LIN {X 0,Y 421.13,Z 404.126,A -85,B 0,C 180,E1 -10185.61,E2 -10185.61} C_VEL
LIN {X 0,Y 421.83,Z 391.614,A -85,B 0,C 180,E1 -10186.266,E2 -10186.266} C_VEL
LIN {X 0,Y 422.346,Z 378.565,A -85,B 0,C 180,E1 -10186.743,E2 -10186.743} C_VEL
LIN {X 0,Y 422.673,Z 363.001,A -85,B 0,C 180,E1 -10187.072,E2 -10187.072} C_VEL
LIN {X 0,Y 423.413,Z 291.136,A -85,B 0,C 180,E1 -10188.331,E2 -10188.331} C_VEL
LIN {X 0,Y 419.56,Z 265.858,A -85,B 0,C 180,E1 -10188.963,E2 -10188.963} C_VEL
LIN {X 0,Y 420.642,Z 248.412,A -85,B 0,C 180,E1 -10192.339,E2 -10192.339} C_VEL
LIN {X 0,Y 421.257,Z 237.979,A -85,B 0,C 180,E1 -10194.387,E2 -10194.387} C_VEL
LIN {X 0,Y 419.001,Z 226.058,A -85,B 0,C 180,E1 -10196.928,E2 -10196.928} C_VEL
LIN {X 0,Y 418.244,Z 222.39,A -85,B 0,C 180,E1 -10197.752,E2 -10197.752} C_VEL
LIN {X 0,Y 418.218,Z 222.388,A -85,B 0,C 180,E1 -10201.01,E2 -10201.01} C_VEL
LIN {X 0,Y 418.219,Z 222.392,A -85,B 0,C 180,E1 -10203.679,E2 -10203.679} C_VEL
LIN {X 0,Y 418.234,Z 222.385,A -85,B 0,C 180,E1 -10207.224,E2 -10207.224} C_VEL
LIN {X 0,Y 418.214,Z 222.386,A -85,B 0,C 180,E1 -10210.948,E2 -10210.948} C_VEL
LIN {X 0,Y 418.164,Z 222.4,A -85,B 0,C 180,E1 -10213.719,E2 -10213.719} C_VEL
LIN {X 0,Y 418.184,Z 222.391,A -85,B 0,C 180,E1 -10216.441,E2 -10216.441} C_VEL
LIN {X 0,Y 418.213,Z 222.388,A -85,B 0,C 180,E1 -10219.13,E2 -10219.13} C_VEL
LIN {X 0,Y 418.23,Z 222.384,A -85,B 0,C 180,E1 -10222.771,E2 -10222.771} C_VEL
LIN {X 0,Y 418.223,Z 222.386,A -85,B 0,C 180,E1 -10226.316,E2 -10226.316} C_VEL
LIN {X 0,Y 418.237,Z 222.39,A -85,B 0,C 180,E1 -10229.723,E2 -10229.723} C_VEL
LIN {X 0,Y 418.197,Z 222.389,A -85,B 0,C 180,E1 -10233.011,E2 -10233.011} C_VEL
LIN {X 0,Y 418.255,Z 222.382,A -85,B 0,C 180,E1 -10236.212,E2 -10236.212} C_VEL
LIN {X 0,Y 418.237,Z 222.387,A -85,B 0,C 180,E1 -10239.332,E2 -10239.332} C_VEL
LIN {X 0,Y 418.261,Z 222.381,A -85,B 0,C 180,E1 -10242.39,E2 -10242.39} C_VEL
LIN {X 0,Y 418.28,Z 222.383,A -85,B 0,C 180,E1 -10245.397,E2 -10245.397} C_VEL
LIN {X 0,Y 418.291,Z 222.377,A -85,B 0,C 180,E1 -10248.363,E2 -10248.363} C_VEL
LIN {X 0,Y 418.441,Z 222.358,A -85,B 0,C 180,E1 -10252.273,E2 -10252.273} C_VEL
LIN {X 0,Y 418.46,Z 222.356,A -85,B 0,C 180,E1 -10254.211,E2 -10254.211} C_VEL
LIN {X 0,Y 418.518,Z 222.35,A -85,B 0,C 180,E1 -10258.07,E2 -10258.07} C_VEL
LIN {X 0,Y 418.393,Z 222.365,A -85,B 0,C 180,E1 -10260.957,E2 -10260.957} C_VEL
LIN {X 0,Y 418.465,Z 222.356,A -85,B 0,C 180,E1 -10262.882,E2 -10262.882} C_VEL
LIN {X 0,Y 418.418,Z 222.361,A -85,B 0,C 180,E1 -10266.746,E2 -10266.746} C_VEL
LIN {X 0,Y 418.307,Z 222.379,A -85,B 0,C 180,E1 -10269.666,E2 -10269.666} C_VEL
LIN {X 0,Y 418.326,Z 222.375,A -85,B 0,C 180,E1 -10272.994,E2 -10272.994} C_VEL
LIN {X 0,Y 418.288,Z 222.378,A -85,B 0,C 180,E1 -10276.729,E2 -10276.729} C_VEL
LIN {X 0,Y 418.244,Z 222.385,A -85,B 0,C 180,E1 -10279.784,E2 -10279.784} C_VEL
LIN {X 0,Y 418.208,Z 222.388,A -85,B 0,C 180,E1 -10282.731,E2 -10282.731} C_VEL
LIN {X 0,Y 418.208,Z 222.389,A -85,B 0,C 180,E1 -10285.9,E2 -10285.9} C_VEL
LIN {X 0,Y 418.231,Z 222.389,A -85,B 0,C 180,E1 -10289.156,E2 -10289.156} C_VEL
LIN {X 0,Y 418.22,Z 222.387,A -85,B 0,C 180,E1 -10292.838,E2 -10292.838} C_VEL
LIN {X 0,Y 418.204,Z 222.387,A -85,B 0,C 180,E1 -10296.232,E2 -10296.232} C_VEL
LIN {X 0,Y 418.208,Z 222.39,A -85,B 0,C 180,E1 -10299.677,E2 -10299.677} C_VEL
LIN {X 0,Y 418.186,Z 222.39,A -85,B 0,C 180,E1 -10302.316,E2 -10302.316} C_VEL
LIN {X 0,Y 418.191,Z 222.394,A -85,B 0,C 180,E1 -10305.104,E2 -10305.104} C_VEL
LIN {X 0,Y 418.191,Z 222.391,A -85,B 0,C 180,E1 -10307.762,E2 -10307.762} C_VEL
LIN {X 0,Y 418.206,Z 222.391,A -85,B 0,C 180,E1 -10311.554,E2 -10311.554} C_VEL
LIN {X 0,Y 418.207,Z 222.394,A -85,B 0,C 180,E1 -10315.155,E2 -10315.155} C_VEL
LIN {X 0,Y 418.191,Z 222.393,A -85,B 0,C 180,E1 -10317.468,E2 -10317.468} C_VEL
LIN {X 0,Y 418.22,Z 222.389,A -85,B 0,C 180,E1 -10320.89,E2 -10320.89} C_VEL
LIN {X 0,Y 418.216,Z 222.386,A -85,B 0,C 180,E1 -10324.093,E2 -10324.093} C_VEL
LIN {X 0,Y 418.218,Z 222.389,A -85,B 0,C 180,E1 -10327.534,E2 -10327.534} C_VEL
LIN {X 0,Y 418.257,Z 222.381,A -85,B 0,C 180,E1 -10330.363,E2 -10330.363} C_VEL
LIN {X 0,Y 418.265,Z 222.384,A -85,B 0,C 180,E1 -10333.403,E2 -10333.403} C_VEL
LIN {X 0,Y 418.293,Z 222.382,A -85,B 0,C 180,E1 -10336.992,E2 -10336.992} C_VEL
LIN {X 0,Y 418.305,Z 222.375,A -85,B 0,C 180,E1 -10340.328,E2 -10340.328} C_VEL
LIN {X 0,Y 418.453,Z 222.362,A -85,B 0,C 180,E1 -10343.248,E2 -10343.248} C_VEL
LIN {X 0,Y 418.286,Z 222.383,A -85,B 0,C 180,E1 -10345.181,E2 -10345.181} C_VEL
LIN {X 0,Y 418.482,Z 222.353,A -85,B 0,C 180,E1 -10348.075,E2 -10348.075} C_VEL
LIN {X 0,Y 418.61,Z 222.337,A -85,B 0,C 180,E1 -10350,E2 -10350} C_VEL
LIN {X 0,Y 418.456,Z 222.362,A -85,B 0,C 180,E1 -10352.888,E2 -10352.888} C_VEL
LIN {X 0,Y 418.479,Z 222.355,A -85,B 0,C 180,E1 -10355.783,E2 -10355.783} C_VEL
LIN {X 0,Y 418.355,Z 222.375,A -85,B 0,C 180,E1 -10358.696,E2 -10358.696} C_VEL
LIN {X 0,Y 418.317,Z 222.57,A -85,B 0,C 180,E1 -10360.772,E2 -10360.772} C_VEL
LIN {X 0,Y 419.131,Z 226.7,A -85,B 0,C 180,E1 -10361.775,E2 -10361.775} C_VEL
LIN {X 0,Y 418.75,Z 229.04,A -85,B 0,C 180,E1 -10362.288,E2 -10362.288} C_VEL
LIN {X 0,Y 416.077,Z 233.116,A -85,B 0,C 180,E1 -10363.077,E2 -10363.077} C_VEL
LIN {X 0,Y 413.78,Z 237.058,A -85,B 0,C 180,E1 -10363.687,E2 -10363.687} C_VEL
LIN {X 0,Y 413.53,Z 239.678,A -85,B 0,C 180,E1 -10363.885,E2 -10363.885} C_VEL
LIN {X 0,Y 413.619,Z 240.251,A -85,B 0,C 180,E1 -10363.905,E2 -10363.905} C_VEL
LIN {X 0,Y 417.073,Z 257.796,A -85,B 0,C 180,E1 -10364.388,E2 -10364.388} C_VEL
LIN {X 0,Y 415.839,Z 344.239,A -85,B 0,C 180,E1 -10365.94,E2 -10365.94} C_VEL
LIN {X 0,Y 415.403,Z 357.444,A -85,B 0,C 180,E1 -10366.367,E2 -10366.367} C_VEL
LIN {X 0,Y 414.936,Z 370.256,A -85,B 0,C 180,E1 -10366.988,E2 -10366.988} C_VEL
LIN {X 0,Y 414.351,Z 382.19,A -85,B 0,C 180,E1 -10367.776,E2 -10367.776} C_VEL
LIN {X 0,Y 413.625,Z 393.478,A -85,B 0,C 180,E1 -10368.735,E2 -10368.735} C_VEL
LIN {X 0,Y 412.878,Z 404.419,A -85,B 0,C 180,E1 -10369.903,E2 -10369.903} C_VEL
LIN {X 0,Y 412.209,Z 412.623,A -85,B 0,C 180,E1 -10370.979,E2 -10370.979} C_VEL
LIN {X 0,Y 411.605,Z 421.45,A -85,B 0,C 180,E1 -10372.403,E2 -10372.403} C_VEL
LIN {X 0,Y 411.011,Z 429.216,A -85,B 0,C 180,E1 -10373.96,E2 -10373.96} C_VEL
LIN {X 0,Y 410.626,Z 434.689,A -85,B 0,C 180,E1 -10375.333,E2 -10375.333} C_VEL
LIN {X 0,Y 410.322,Z 440.075,A -85,B 0,C 180,E1 -10377.063,E2 -10377.063} C_VEL
LIN {X 0,Y 410.119,Z 443.73,A -85,B 0,C 180,E1 -10378.673,E2 -10378.673} C_VEL
LIN {X 0,Y 409.947,Z 445.615,A -85,B 0,C 180,E1 -10379.812,E2 -10379.812} C_VEL
LIN {X 0,Y 409.835,Z 446.965,A -85,B 0,C 180,E1 -10380.989,E2 -10380.989} C_VEL
LIN {X 0,Y 409.79,Z 447.919,A -85,B 0,C 180,E1 -10382.837,E2 -10382.837} C_VEL
LIN {X 0,Y 409.805,Z 447.533,A -85,B 0,C 180,E1 -10384.61,E2 -10384.61} C_VEL
LIN {X 0,Y 409.934,Z 445.905,A -85,B 0,C 180,E1 -10386.329,E2 -10386.329} C_VEL
LIN {X 0,Y 410.214,Z 442.914,A -85,B 0,C 180,E1 -10388.079,E2 -10388.079} C_VEL
LIN {X 0,Y 410.418,Z 439.178,A -85,B 0,C 180,E1 -10389.607,E2 -10389.607} C_VEL
LIN {X 0,Y 410.771,Z 434.092,A -85,B 0,C 180,E1 -10391.178,E2 -10391.178} C_VEL
LIN {X 0,Y 411.289,Z 427.699,A -85,B 0,C 180,E1 -10392.724,E2 -10392.724} C_VEL
LIN {X 0,Y 411.967,Z 419.754,A -85,B 0,C 180,E1 -10394.245,E2 -10394.245} C_VEL
LIN {X 0,Y 412.732,Z 410.523,A -85,B 0,C 180,E1 -10395.656,E2 -10395.656} C_VEL
LIN {X 0,Y 413.412,Z 401.414,A -85,B 0,C 180,E1 -10396.79,E2 -10396.79} C_VEL
LIN {X 0,Y 414.188,Z 391.232,A -85,B 0,C 180,E1 -10397.822,E2 -10397.822} C_VEL
LIN {X 0,Y 414.926,Z 379.902,A -85,B 0,C 180,E1 -10398.732,E2 -10398.732} C_VEL
LIN {X 0,Y 415.566,Z 367.793,A -85,B 0,C 180,E1 -10399.483,E2 -10399.483} C_VEL
LIN {X 0,Y 416.066,Z 355.316,A -85,B 0,C 180,E1 -10400.051,E2 -10400.051} C_VEL
LIN {X 0,Y 416.391,Z 342.292,A -85,B 0,C 180,E1 -10400.433,E2 -10400.433} C_VEL
LIN {X 0,Y 417.621,Z 257.355,A -85,B 0,C 180,E1 -10401.968,E2 -10401.968} C_VEL
LIN {X 0,Y 413.763,Z 239.192,A -85,B 0,C 180,E1 -10402.513,E2 -10402.513} C_VEL
LIN {X 0,Y 413.33,Z 237.054,A -85,B 0,C 180,E1 -10402.61,E2 -10402.61} C_VEL
LIN {X 0,Y 413.225,Z 233.046,A -85,B 0,C 180,E1 -10403.478,E2 -10403.478} C_VEL
LIN {X 0,Y 411.22,Z 223.265,A -85,B 0,C 180,E1 -10405.751,E2 -10405.751} C_VEL
LIN {X 0,Y 411.162,Z 223.272,A -85,B 0,C 180,E1 -10409.159,E2 -10409.159} C_VEL
LIN {X 0,Y 411.228,Z 223.26,A -85,B 0,C 180,E1 -10412.528,E2 -10412.528} C_VEL
LIN {X 0,Y 411.197,Z 223.263,A -85,B 0,C 180,E1 -10415.79,E2 -10415.79} C_VEL
LIN {X 0,Y 411.169,Z 223.273,A -85,B 0,C 180,E1 -10418.972,E2 -10418.972} C_VEL
LIN {X 0,Y 411.228,Z 223.261,A -85,B 0,C 180,E1 -10422.091,E2 -10422.091} C_VEL
LIN {X 0,Y 411.239,Z 223.259,A -85,B 0,C 180,E1 -10425.153,E2 -10425.153} C_VEL
LIN {X 0,Y 411.28,Z 223.251,A -85,B 0,C 180,E1 -10428.174,E2 -10428.174} C_VEL
LIN {X 0,Y 411.422,Z 223.232,A -85,B 0,C 180,E1 -10432.197,E2 -10432.197} C_VEL
LIN {X 0,Y 411.432,Z 223.233,A -85,B 0,C 180,E1 -10434.123,E2 -10434.123} C_VEL
LIN {X 0,Y 411.498,Z 223.222,A -85,B 0,C 180,E1 -10438.048,E2 -10438.048} C_VEL
LIN {X 0,Y 411.625,Z 223.208,A -85,B 0,C 180,E1 -10440.006,E2 -10440.006} C_VEL
LIN {X 0,Y 411.425,Z 223.235,A -85,B 0,C 180,E1 -10442.943,E2 -10442.943} C_VEL
LIN {X 0,Y 411.424,Z 223.235,A -85,B 0,C 180,E1 -10446.873,E2 -10446.873} C_VEL
LIN {X 0,Y 411.278,Z 223.247,A -85,B 0,C 180,E1 -10449.844,E2 -10449.844} C_VEL
LIN {X 0,Y 411.302,Z 223.247,A -85,B 0,C 180,E1 -10453.109,E2 -10453.109} C_VEL
LIN {X 0,Y 411.257,Z 223.256,A -85,B 0,C 180,E1 -10456.894,E2 -10456.894} C_VEL
LIN {X 0,Y 411.232,Z 223.257,A -85,B 0,C 180,E1 -10459.991,E2 -10459.991} C_VEL
LIN {X 0,Y 411.188,Z 223.262,A -85,B 0,C 180,E1 -10463.153,E2 -10463.153} C_VEL
LIN {X 0,Y 411.167,Z 223.265,A -85,B 0,C 180,E1 -10466.39,E2 -10466.39} C_VEL
LIN {X 0,Y 411.2,Z 223.259,A -85,B 0,C 180,E1 -10469.717,E2 -10469.717} C_VEL
LIN {X 0,Y 411.209,Z 223.257,A -85,B 0,C 180,E1 -10473.16,E2 -10473.16} C_VEL
LIN {X 0,Y 411.194,Z 223.264,A -85,B 0,C 180,E1 -10476.555,E2 -10476.555} C_VEL
LIN {X 0,Y 411.169,Z 223.265,A -85,B 0,C 180,E1 -10479.722,E2 -10479.722} C_VEL
LIN {X 0,Y 411.131,Z 223.273,A -85,B 0,C 180,E1 -10483.144,E2 -10483.144} C_VEL
LIN {X 0,Y 411.156,Z 223.272,A -85,B 0,C 180,E1 -10485.887,E2 -10485.887} C_VEL
LIN {X 0,Y 411.164,Z 223.267,A -85,B 0,C 180,E1 -10489.495,E2 -10489.495} C_VEL
LIN {X 0,Y 411.185,Z 223.269,A -85,B 0,C 180,E1 -10492.027,E2 -10492.027} C_VEL
LIN {X 0,Y 411.208,Z 223.262,A -85,B 0,C 180,E1 -10495.127,E2 -10495.127} C_VEL
LIN {X 0,Y 411.163,Z 223.276,A -85,B 0,C 180,E1 -10498.004,E2 -10498.004} C_VEL
LIN {X 0,Y 411.183,Z 223.271,A -85,B 0,C 180,E1 -10501.408,E2 -10501.408} C_VEL
LIN {X 0,Y 411.184,Z 223.35,A -85,B 0,C 180,E1 -10502.034,E2 -10502.034} C_VEL
LIN {X 0,Y 413.567,Z 234.523,A -85,B 0,C 180,E1 -10504.482,E2 -10504.482} C_VEL
LIN {X 0,Y 414.356,Z 240.401,A -85,B 0,C 180,E1 -10505.714,E2 -10505.714} C_VEL
LIN {X 0,Y 413.278,Z 256.322,A -85,B 0,C 180,E1 -10508.816,E2 -10508.816} C_VEL
LIN {X 0,Y 412.823,Z 264.691,A -85,B 0,C 180,E1 -10510.435,E2 -10510.435} C_VEL
LIN {X 0,Y 416.982,Z 290.686,A -85,B 0,C 180,E1 -10511.14,E2 -10511.14} C_VEL
LIN {X 0,Y 417.212,Z 298.733,A -85,B 0,C 180,E1 -10511.302,E2 -10511.302} C_VEL
LIN {X 0,Y 416.178,Z 374.289,A -85,B 0,C 180,E1 -10512.685,E2 -10512.685} C_VEL
LIN {X 0,Y 415.578,Z 387.154,A -85,B 0,C 180,E1 -10513.103,E2 -10513.103} C_VEL
LIN {X 0,Y 414.874,Z 399.702,A -85,B 0,C 180,E1 -10513.706,E2 -10513.706} C_VEL
LIN {X 0,Y 414.051,Z 411.72,A -85,B 0,C 180,E1 -10514.495,E2 -10514.495} C_VEL
LIN {X 0,Y 413.284,Z 423.495,A -85,B 0,C 180,E1 -10515.499,E2 -10515.499} C_VEL
LIN {X 0,Y 412.488,Z 433.635,A -85,B 0,C 180,E1 -10516.577,E2 -10516.577} C_VEL
LIN {X 0,Y 411.885,Z 442.149,A -85,B 0,C 180,E1 -10517.685,E2 -10517.685} C_VEL
LIN {X 0,Y 411.061,Z 451.381,A -85,B 0,C 180,E1 -10519.16,E2 -10519.16} C_VEL
LIN {X 0,Y 410.606,Z 458.83,A -85,B 0,C 180,E1 -10520.642,E2 -10520.642} C_VEL
LIN {X 0,Y 410.279,Z 464.815,A -85,B 0,C 180,E1 -10522.124,E2 -10522.124} C_VEL
LIN {X 0,Y 410.036,Z 470.092,A -85,B 0,C 180,E1 -10523.803,E2 -10523.803} C_VEL
LIN {X 0,Y 410.016,Z 473.156,A -85,B 0,C 180,E1 -10525.084,E2 -10525.084} C_VEL
LIN {X 0,Y 409.938,Z 475.002,A -85,B 0,C 180,E1 -10526.068,E2 -10526.068} C_VEL
LIN {X 0,Y 410.003,Z 477.393,A -85,B 0,C 180,E1 -10528.035,E2 -10528.035} C_VEL
LIN {X 0,Y 409.945,Z 477.993,A -85,B 0,C 180,E1 -10529.018,E2 -10529.018} C_VEL
LIN {X 0,Y 409.935,Z 478.174,A -85,B 0,C 180,E1 -10530,E2 -10530} C_VEL
LIN {X 0,Y 410.003,Z 477.303,A -85,B 0,C 180,E1 -10531.965,E2 -10531.965} C_VEL
LIN {X 0,Y 409.937,Z 476.274,A -85,B 0,C 180,E1 -10532.948,E2 -10532.948} C_VEL
LIN {X 0,Y 409.938,Z 474.809,A -85,B 0,C 180,E1 -10533.932,E2 -10533.932} C_VEL
LIN {X 0,Y 409.996,Z 471.793,A -85,B 0,C 180,E1 -10535.41,E2 -10535.41} C_VEL
LIN {X 0,Y 410.175,Z 467.711,A -85,B 0,C 180,E1 -10536.888,E2 -10536.888} C_VEL
LIN {X 0,Y 410.432,Z 461.424,A -85,B 0,C 180,E1 -10538.617,E2 -10538.617} C_VEL
LIN {X 0,Y 410.839,Z 454.576,A -85,B 0,C 180,E1 -10540.098,E2 -10540.098} C_VEL
LIN {X 0,Y 411.291,Z 447.586,A -85,B 0,C 180,E1 -10541.333,E2 -10541.333} C_VEL
LIN {X 0,Y 411.942,Z 439.171,A -85,B 0,C 180,E1 -10542.563,E2 -10542.563} C_VEL
LIN {X 0,Y 412.67,Z 428.8,A -85,B 0,C 180,E1 -10543.793,E2 -10543.793} C_VEL
LIN {X 0,Y 413.416,Z 417.096,A -85,B 0,C 180,E1 -10544.899,E2 -10544.899} C_VEL
LIN {X 0,Y 414.136,Z 405.504,A -85,B 0,C 180,E1 -10545.755,E2 -10545.755} C_VEL
LIN {X 0,Y 414.84,Z 393.49,A -85,B 0,C 180,E1 -10546.422,E2 -10546.422} C_VEL
LIN {X 0,Y 415.45,Z 380.532,A -85,B 0,C 180,E1 -10546.934,E2 -10546.934} C_VEL
LIN {X 0,Y 415.772,Z 368.445,A -85,B 0,C 180,E1 -10547.237,E2 -10547.237} C_VEL
LIN {X 0,Y 416.664,Z 292.238,A -85,B 0,C 180,E1 -10548.594,E2 -10548.594} C_VEL
LIN {X 0,Y 412.611,Z 265.599,A -85,B 0,C 180,E1 -10549.276,E2 -10549.276} C_VEL
LIN {X 0,Y 413.796,Z 248.074,A -85,B 0,C 180,E1 -10552.73,E2 -10552.73} C_VEL
LIN {X 0,Y 414.263,Z 238.927,A -85,B 0,C 180,E1 -10554.559,E2 -10554.559} C_VEL
LIN {X 0,Y 411.887,Z 226.556,A -85,B 0,C 180,E1 -10557.25,E2 -10557.25} C_VEL
LIN {X 0,Y 411.196,Z 223.266,A -85,B 0,C 180,E1 -10558.035,E2 -10558.035} C_VEL
LIN {X 0,Y 411.164,Z 223.268,A -85,B 0,C 180,E1 -10561.274,E2 -10561.274} C_VEL
LIN {X 0,Y 411.169,Z 223.265,A -85,B 0,C 180,E1 -10564.336,E2 -10564.336} C_VEL
LIN {X 0,Y 411.187,Z 223.262,A -85,B 0,C 180,E1 -10566.741,E2 -10566.741} C_VEL
LIN {X 0,Y 411.171,Z 223.27,A -85,B 0,C 180,E1 -10569.716,E2 -10569.716} C_VEL
LIN {X 0,Y 411.113,Z 223.272,A -85,B 0,C 180,E1 -10573.14,E2 -10573.14} C_VEL
LIN {X 0,Y 411.151,Z 223.272,A -85,B 0,C 180,E1 -10575.882,E2 -10575.882} C_VEL
LIN {X 0,Y 411.163,Z 223.269,A -85,B 0,C 180,E1 -10579.489,E2 -10579.489} C_VEL
LIN {X 0,Y 411.18,Z 223.266,A -85,B 0,C 180,E1 -10582.02,E2 -10582.02} C_VEL
LIN {X 0,Y 411.191,Z 223.262,A -85,B 0,C 180,E1 -10585.123,E2 -10585.123} C_VEL
LIN {X 0,Y 411.157,Z 223.269,A -85,B 0,C 180,E1 -10587.998,E2 -10587.998} C_VEL
LIN {X 0,Y 411.17,Z 223.268,A -85,B 0,C 180,E1 -10591.402,E2 -10591.402} C_VEL
LIN {X 0,Y 411.19,Z 223.262,A -85,B 0,C 180,E1 -10594.937,E2 -10594.937} C_VEL
LIN {X 0,Y 411.201,Z 223.264,A -85,B 0,C 180,E1 -10597.909,E2 -10597.909} C_VEL
LIN {X 0,Y 411.187,Z 223.263,A -85,B 0,C 180,E1 -10601.045,E2 -10601.045} C_VEL
LIN {X 0,Y 411.238,Z 223.257,A -85,B 0,C 180,E1 -10604.126,E2 -10604.126} C_VEL
LIN {X 0,Y 411.298,Z 223.25,A -85,B 0,C 180,E1 -10607.161,E2 -10607.161} C_VEL
LIN {X 0,Y 411.265,Z 223.253,A -85,B 0,C 180,E1 -10610.156,E2 -10610.156} C_VEL
LIN {X 0,Y 411.383,Z 223.24,A -85,B 0,C 180,E1 -10613.127,E2 -10613.127} C_VEL
LIN {X 0,Y 411.272,Z 223.253,A -85,B 0,C 180,E1 -10615.093,E2 -10615.093} C_VEL
LIN {X 0,Y 411.487,Z 223.226,A -85,B 0,C 180,E1 -10618.037,E2 -10618.037} C_VEL
LIN {X 0,Y 411.492,Z 223.226,A -85,B 0,C 180,E1 -10621.952,E2 -10621.952} C_VEL
LIN {X 0,Y 411.364,Z 223.239,A -85,B 0,C 180,E1 -10626.5,E2 -10626.5} C_VEL
LIN {X 0,Y 411.291,Z 223.25,A -85,B 0,C 180,E1 -10628.84,E2 -10628.84} C_VEL
LIN {X 0,Y 411.26,Z 223.255,A -85,B 0,C 180,E1 -10631.827,E2 -10631.827} C_VEL
LIN {X 0,Y 411.234,Z 223.257,A -85,B 0,C 180,E1 -10634.847,E2 -10634.847} C_VEL
LIN {X 0,Y 411.22,Z 223.259,A -85,B 0,C 180,E1 -10637.91,E2 -10637.91} C_VEL
LIN {X 0,Y 411.169,Z 223.267,A -85,B 0,C 180,E1 -10641.028,E2 -10641.028} C_VEL
LIN {X 0,Y 411.179,Z 223.263,A -85,B 0,C 180,E1 -10644.211,E2 -10644.211} C_VEL
LIN {X 0,Y 411.21,Z 223.265,A -85,B 0,C 180,E1 -10647.473,E2 -10647.473} C_VEL
LIN {X 0,Y 411.154,Z 223.267,A -85,B 0,C 180,E1 -10650.842,E2 -10650.842} C_VEL
LIN {X 0,Y 411.167,Z 223.264,A -85,B 0,C 180,E1 -10654.328,E2 -10654.328} C_VEL
LIN {X 0,Y 411.154,Z 223.267,A -85,B 0,C 180,E1 -10657.968,E2 -10657.968} C_VEL
LIN {X 0,Y 411.139,Z 223.268,A -85,B 0,C 180,E1 -10660.499,E2 -10660.499} C_VEL
LIN {X 0,Y 411.132,Z 223.274,A -85,B 0,C 180,E1 -10663.128,E2 -10663.128} C_VEL
LIN {X 0,Y 411.121,Z 223.271,A -85,B 0,C 180,E1 -10665.876,E2 -10665.876} C_VEL
LIN {X 0,Y 411.114,Z 223.273,A -85,B 0,C 180,E1 -10668.767,E2 -10668.767} C_VEL
LIN {X 0,Y 411.148,Z 223.267,A -85,B 0,C 180,E1 -10672.022,E2 -10672.022} C_VEL
LIN {X 0,Y 411.152,Z 223.268,A -85,B 0,C 180,E1 -10675.662,E2 -10675.662} C_VEL
LIN {X 0,Y 411.142,Z 223.274,A -85,B 0,C 180,E1 -10679.149,E2 -10679.149} C_VEL
LIN {X 0,Y 411.203,Z 223.26,A -85,B 0,C 180,E1 -10682.519,E2 -10682.519} C_VEL
LIN {X 0,Y 411.173,Z 223.264,A -85,B 0,C 180,E1 -10685.782,E2 -10685.782} C_VEL
LIN {X 0,Y 411.179,Z 223.268,A -85,B 0,C 180,E1 -10688.965,E2 -10688.965} C_VEL
LIN {X 0,Y 411.195,Z 223.261,A -85,B 0,C 180,E1 -10692.083,E2 -10692.083} C_VEL
LIN {X 0,Y 411.205,Z 223.267,A -85,B 0,C 180,E1 -10695.146,E2 -10695.146} C_VEL
LIN {X 0,Y 411.24,Z 223.255,A -85,B 0,C 180,E1 -10698.166,E2 -10698.166} C_VEL
LIN {X 0,Y 411.419,Z 223.233,A -85,B 0,C 180,E1 -10702.146,E2 -10702.146} C_VEL
LIN {X 0,Y 411.438,Z 223.23,A -85,B 0,C 180,E1 -10704.118,E2 -10704.118} C_VEL
LIN {X 0,Y 411.451,Z 223.229,A -85,B 0,C 180,E1 -10708.042,E2 -10708.042} C_VEL
LIN {X 0,Y 411.58,Z 223.213,A -85,B 0,C 180,E1 -10710,E2 -10710} C_VEL
LIN {X 0,Y 411.411,Z 223.24,A -85,B 0,C 180,E1 -10712.937,E2 -10712.937} C_VEL
LIN {X 0,Y 411.438,Z 223.232,A -85,B 0,C 180,E1 -10715.882,E2 -10715.882} C_VEL
LIN {X 0,Y 411.307,Z 223.254,A -85,B 0,C 180,E1 -10718.846,E2 -10718.846} C_VEL
LIN {X 0,Y 411.287,Z 223.317,A -85,B 0,C 180,E1 -10720.522,E2 -10720.522} C_VEL
LIN {X 0,Y 412.947,Z 232.58,A -85,B 0,C 180,E1 -10722.782,E2 -10722.782} C_VEL
LIN {X 0,Y 412.986,Z 237.016,A -85,B 0,C 180,E1 -10723.807,E2 -10723.807} C_VEL
LIN {X 0,Y 413.619,Z 240.251,A -85,B 0,C 180,E1 -10723.905,E2 -10723.905} C_VEL
LIN {X 0,Y 414.059,Z 246.078,A -85,B 0,C 180,E1 -10724.034,E2 -10724.034} C_VEL
LIN {X 0,Y 413.405,Z 251.982,A -85,B 0,C 180,E1 -10724.115,E2 -10724.115} C_VEL
LIN {X 0,Y 410.319,Z 267.779,A -85,B 0,C 180,E1 -10724.271,E2 -10724.271} C_VEL
LIN {X 0,Y 410.095,Z 271.776,A -85,B 0,C 180,E1 -10724.336,E2 -10724.336} C_VEL
LIN {X 0,Y 409.001,Z 345.346,A -85,B 0,C 180,E1 -10725.692,E2 -10725.692} C_VEL
LIN {X 0,Y 408.574,Z 358.46,A -85,B 0,C 180,E1 -10726.135,E2 -10726.135} C_VEL
LIN {X 0,Y 408.079,Z 371.07,A -85,B 0,C 180,E1 -10726.766,E2 -10726.766} C_VEL
LIN {X 0,Y 407.443,Z 382.88,A -85,B 0,C 180,E1 -10727.569,E2 -10727.569} C_VEL
LIN {X 0,Y 406.719,Z 393.807,A -85,B 0,C 180,E1 -10728.516,E2 -10728.516} C_VEL
LIN {X 0,Y 405.976,Z 403.835,A -85,B 0,C 180,E1 -10729.597,E2 -10729.597} C_VEL
LIN {X 0,Y 405.288,Z 412.117,A -85,B 0,C 180,E1 -10730.682,E2 -10730.682} C_VEL
LIN {X 0,Y 404.704,Z 419.962,A -85,B 0,C 180,E1 -10731.923,E2 -10731.923} C_VEL
LIN {X 0,Y 404.18,Z 426.642,A -85,B 0,C 180,E1 -10733.198,E2 -10733.198} C_VEL
LIN {X 0,Y 403.77,Z 433.031,A -85,B 0,C 180,E1 -10734.691,E2 -10734.691} C_VEL
LIN {X 0,Y 403.336,Z 438.668,A -85,B 0,C 180,E1 -10736.38,E2 -10736.38} C_VEL
LIN {X 0,Y 403.146,Z 442.914,A -85,B 0,C 180,E1 -10738.078,E2 -10738.078} C_VEL
LIN {X 0,Y 402.931,Z 445.199,A -85,B 0,C 180,E1 -10739.313,E2 -10739.313} C_VEL
LIN {X 0,Y 402.729,Z 447.451,A -85,B 0,C 180,E1 -10741.246,E2 -10741.246} C_VEL
LIN {X 0,Y 402.705,Z 448.227,A -85,B 0,C 180,E1 -10743.118,E2 -10743.118} C_VEL
LIN {X 0,Y 402.716,Z 447.632,A -85,B 0,C 180,E1 -10744.908,E2 -10744.908} C_VEL
LIN {X 0,Y 402.883,Z 445.816,A -85,B 0,C 180,E1 -10746.651,E2 -10746.651} C_VEL
LIN {X 0,Y 403.152,Z 442.849,A -85,B 0,C 180,E1 -10748.342,E2 -10748.342} C_VEL
LIN {X 0,Y 403.483,Z 438.351,A -85,B 0,C 180,E1 -10750.125,E2 -10750.125} C_VEL
LIN {X 0,Y 403.908,Z 432.676,A -85,B 0,C 180,E1 -10751.789,E2 -10751.789} C_VEL
LIN {X 0,Y 404.565,Z 425.055,A -85,B 0,C 180,E1 -10753.517,E2 -10753.517} C_VEL
LIN {X 0,Y 405.247,Z 417.384,A -85,B 0,C 180,E1 -10754.904,E2 -10754.904} C_VEL
LIN {X 0,Y 405.964,Z 408.684,A -85,B 0,C 180,E1 -10756.185,E2 -10756.185} C_VEL
LIN {X 0,Y 406.884,Z 397.812,A -85,B 0,C 180,E1 -10757.469,E2 -10757.469} C_VEL
LIN {X 0,Y 407.612,Z 387.993,A -85,B 0,C 180,E1 -10758.404,E2 -10758.404} C_VEL
LIN {X 0,Y 408.343,Z 377.279,A -85,B 0,C 180,E1 -10759.223,E2 -10759.223} C_VEL
LIN {X 0,Y 408.928,Z 366.141,A -85,B 0,C 180,E1 -10759.887,E2 -10759.887} C_VEL
LIN {X 0,Y 409.414,Z 353.346,A -85,B 0,C 180,E1 -10760.437,E2 -10760.437} C_VEL
LIN {X 0,Y 409.725,Z 340.434,A -85,B 0,C 180,E1 -10760.792,E2 -10760.792} C_VEL
LIN {X 0,Y 410.991,Z 258.784,A -85,B 0,C 180,E1 -10762.285,E2 -10762.285} C_VEL
LIN {X 0,Y 407.347,Z 241.288,A -85,B 0,C 180,E1 -10762.824,E2 -10762.824} C_VEL
LIN {X 0,Y 406.479,Z 237.409,A -85,B 0,C 180,E1 -10762.964,E2 -10762.964} C_VEL
LIN {X 0,Y 406.045,Z 233.008,A -85,B 0,C 180,E1 -10763.96,E2 -10763.96} C_VEL
LIN {X 0,Y 404.156,Z 224.144,A -85,B 0,C 180,E1 -10766.085,E2 -10766.085} C_VEL
LIN {X 0,Y 404.119,Z 224.148,A -85,B 0,C 180,E1 -10769.721,E2 -10769.721} C_VEL
LIN {X 0,Y 404.164,Z 224.143,A -85,B 0,C 180,E1 -10773.129,E2 -10773.129} C_VEL
LIN {X 0,Y 404.147,Z 224.143,A -85,B 0,C 180,E1 -10775.34,E2 -10775.34} C_VEL
LIN {X 0,Y 404.111,Z 224.147,A -85,B 0,C 180,E1 -10778.586,E2 -10778.586} C_VEL
LIN {X 0,Y 404.185,Z 224.138,A -85,B 0,C 180,E1 -10781.768,E2 -10781.768} C_VEL
LIN {X 0,Y 404.185,Z 224.139,A -85,B 0,C 180,E1 -10784.888,E2 -10784.888} C_VEL
LIN {X 0,Y 404.251,Z 224.126,A -85,B 0,C 180,E1 -10787.965,E2 -10787.965} C_VEL
LIN {X 0,Y 404.25,Z 224.128,A -85,B 0,C 180,E1 -10791.004,E2 -10791.004} C_VEL
LIN {X 0,Y 404.382,Z 224.111,A -85,B 0,C 180,E1 -10794.02,E2 -10794.02} C_VEL
LIN {X 0,Y 404.467,Z 224.098,A -85,B 0,C 180,E1 -10798.014,E2 -10798.014} C_VEL
LIN {X 0,Y 404.594,Z 224.084,A -85,B 0,C 180,E1 -10800.006,E2 -10800.006} C_VEL
LIN {X 0,Y 404.385,Z 224.113,A -85,B 0,C 180,E1 -10802.994,E2 -10802.994} C_VEL
LIN {X 0,Y 404.375,Z 224.114,A -85,B 0,C 180,E1 -10806.993,E2 -10806.993} C_VEL
LIN {X 0,Y 404.242,Z 224.131,A -85,B 0,C 180,E1 -10811.03,E2 -10811.03} C_VEL
LIN {X 0,Y 404.207,Z 224.131,A -85,B 0,C 180,E1 -10814.093,E2 -10814.093} C_VEL
LIN {X 0,Y 404.202,Z 224.132,A -85,B 0,C 180,E1 -10817.197,E2 -10817.197} C_VEL
LIN {X 0,Y 404.165,Z 224.14,A -85,B 0,C 180,E1 -10820.356,E2 -10820.356} C_VEL
LIN {X 0,Y 404.149,Z 224.137,A -85,B 0,C 180,E1 -10823.58,E2 -10823.58} C_VEL
LIN {X 0,Y 404.101,Z 224.146,A -85,B 0,C 180,E1 -10826.888,E2 -10826.888} C_VEL
LIN {X 0,Y 404.147,Z 224.139,A -85,B 0,C 180,E1 -10830.29,E2 -10830.29} C_VEL
LIN {X 0,Y 404.143,Z 224.137,A -85,B 0,C 180,E1 -10833.817,E2 -10833.817} C_VEL
LIN {X 0,Y 404.136,Z 224.142,A -85,B 0,C 180,E1 -10836.877,E2 -10836.877} C_VEL
LIN {X 0,Y 404.125,Z 224.144,A -85,B 0,C 180,E1 -10840.078,E2 -10840.078} C_VEL
LIN {X 0,Y 404.088,Z 224.151,A -85,B 0,C 180,E1 -10843.076,E2 -10843.076} C_VEL
LIN {X 0,Y 404.114,Z 224.15,A -85,B 0,C 180,E1 -10845.923,E2 -10845.923} C_VEL
LIN {X 0,Y 404.106,Z 224.15,A -85,B 0,C 180,E1 -10848.635,E2 -10848.635} C_VEL
LIN {X 0,Y 404.142,Z 224.142,A -85,B 0,C 180,E1 -10851.499,E2 -10851.499} C_VEL
LIN {X 0,Y 404.179,Z 224.139,A -85,B 0,C 180,E1 -10854.985,E2 -10854.985} C_VEL
LIN {X 0,Y 404.141,Z 224.149,A -85,B 0,C 180,E1 -10858.447,E2 -10858.447} C_VEL
LIN {X 0,Y 404.165,Z 224.218,A -85,B 0,C 180,E1 -10861.717,E2 -10861.717} C_VEL
LIN {X 0,Y 406.692,Z 236.252,A -85,B 0,C 180,E1 -10864.405,E2 -10864.405} C_VEL
LIN {X 0,Y 407.447,Z 241.593,A -85,B 0,C 180,E1 -10865.546,E2 -10865.546} C_VEL
LIN {X 0,Y 406.417,Z 256.178,A -85,B 0,C 180,E1 -10868.441,E2 -10868.441} C_VEL
LIN {X 0,Y 405.946,Z 264.397,A -85,B 0,C 180,E1 -10870.06,E2 -10870.06} C_VEL
LIN {X 0,Y 410.164,Z 290.345,A -85,B 0,C 180,E1 -10870.789,E2 -10870.789} C_VEL
LIN {X 0,Y 410.55,Z 295.777,A -85,B 0,C 180,E1 -10870.913,E2 -10870.913} C_VEL
LIN {X 0,Y 409.461,Z 373.623,A -85,B 0,C 180,E1 -10872.36,E2 -10872.36} C_VEL
LIN {X 0,Y 408.849,Z 386.608,A -85,B 0,C 180,E1 -10872.784,E2 -10872.784} C_VEL
LIN {X 0,Y 408.076,Z 399.775,A -85,B 0,C 180,E1 -10873.427,E2 -10873.427} C_VEL
LIN {X 0,Y 407.206,Z 411.685,A -85,B 0,C 180,E1 -10874.227,E2 -10874.227} C_VEL
LIN {X 0,Y 406.397,Z 423.402,A -85,B 0,C 180,E1 -10875.248,E2 -10875.248} C_VEL
LIN {X 0,Y 405.577,Z 433.536,A -85,B 0,C 180,E1 -10876.348,E2 -10876.348} C_VEL
LIN {X 0,Y 404.78,Z 443.633,A -85,B 0,C 180,E1 -10877.72,E2 -10877.72} C_VEL
LIN {X 0,Y 403.951,Z 452.56,A -85,B 0,C 180,E1 -10879.221,E2 -10879.221} C_VEL
LIN {X 0,Y 403.493,Z 459.734,A -85,B 0,C 180,E1 -10880.729,E2 -10880.729} C_VEL
LIN {X 0,Y 403.14,Z 466.288,A -85,B 0,C 180,E1 -10882.487,E2 -10882.487} C_VEL
LIN {X 0,Y 402.913,Z 470.62,A -85,B 0,C 180,E1 -10883.993,E2 -10883.993} C_VEL
LIN {X 0,Y 402.925,Z 472.924,A -85,B 0,C 180,E1 -10884.997,E2 -10884.997} C_VEL
LIN {X 0,Y 402.858,Z 474.761,A -85,B 0,C 180,E1 -10885.999,E2 -10885.999} C_VEL
LIN {X 0,Y 402.914,Z 477.143,A -85,B 0,C 180,E1 -10888.001,E2 -10888.001} C_VEL
LIN {X 0,Y 402.873,Z 477.739,A -85,B 0,C 180,E1 -10889.001,E2 -10889.001} C_VEL
LIN {X 0,Y 402.86,Z 477.909,A -85,B 0,C 180,E1 -10890,E2 -10890} C_VEL
LIN {X 0,Y 402.873,Z 477.663,A -85,B 0,C 180,E1 -10891,E2 -10891} C_VEL
LIN {X 0,Y 402.914,Z 477.027,A -85,B 0,C 180,E1 -10891.999,E2 -10891.999} C_VEL
LIN {X 0,Y 402.837,Z 475.991,A -85,B 0,C 180,E1 -10893,E2 -10893} C_VEL
LIN {X 0,Y 402.858,Z 474.514,A -85,B 0,C 180,E1 -10894.001,E2 -10894.001} C_VEL
LIN {X 0,Y 402.896,Z 471.482,A -85,B 0,C 180,E1 -10895.505,E2 -10895.505} C_VEL
LIN {X 0,Y 403.087,Z 467.384,A -85,B 0,C 180,E1 -10897.01,E2 -10897.01} C_VEL
LIN {X 0,Y 403.384,Z 461.08,A -85,B 0,C 180,E1 -10898.769,E2 -10898.769} C_VEL
LIN {X 0,Y 403.784,Z 454.209,A -85,B 0,C 180,E1 -10900.277,E2 -10900.277} C_VEL
LIN {X 0,Y 404.312,Z 447.199,A -85,B 0,C 180,E1 -10901.531,E2 -10901.531} C_VEL
LIN {X 0,Y 404.953,Z 438.754,A -85,B 0,C 180,E1 -10902.784,E2 -10902.784} C_VEL
LIN {X 0,Y 405.696,Z 428.33,A -85,B 0,C 180,E1 -10904.035,E2 -10904.035} C_VEL
LIN {X 0,Y 406.544,Z 416.585,A -85,B 0,C 180,E1 -10905.157,E2 -10905.157} C_VEL
LIN {X 0,Y 407.284,Z 404.895,A -85,B 0,C 180,E1 -10906.027,E2 -10906.027} C_VEL
LIN {X 0,Y 408.019,Z 392.774,A -85,B 0,C 180,E1 -10906.704,E2 -10906.704} C_VEL
LIN {X 0,Y 408.617,Z 379.633,A -85,B 0,C 180,E1 -10907.226,E2 -10907.226} C_VEL
LIN {X 0,Y 408.953,Z 367.023,A -85,B 0,C 180,E1 -10907.534,E2 -10907.534} C_VEL
LIN {X 0,Y 409.823,Z 292.532,A -85,B 0,C 180,E1 -10908.885,E2 -10908.885} C_VEL
LIN {X 0,Y 405.707,Z 265.348,A -85,B 0,C 180,E1 -10909.597,E2 -10909.597} C_VEL
LIN {X 0,Y 406.921,Z 247.707,A -85,B 0,C 180,E1 -10913.136,E2 -10913.136} C_VEL
LIN {X 0,Y 407.385,Z 241.186,A -85,B 0,C 180,E1 -10914.458,E2 -10914.458} C_VEL
LIN {X 0,Y 405.976,Z 232.952,A -85,B 0,C 180,E1 -10916.258,E2 -10916.258} C_VEL
LIN {X 0,Y 404.141,Z 224.145,A -85,B 0,C 180,E1 -10918.285,E2 -10918.285} C_VEL
LIN {X 0,Y 404.125,Z 224.146,A -85,B 0,C 180,E1 -10921.549,E2 -10921.549} C_VEL
LIN {X 0,Y 404.133,Z 224.141,A -85,B 0,C 180,E1 -10925.02,E2 -10925.02} C_VEL
LIN {X 0,Y 404.137,Z 224.14,A -85,B 0,C 180,E1 -10928.5,E2 -10928.5} C_VEL
LIN {X 0,Y 404.093,Z 224.15,A -85,B 0,C 180,E1 -10931.59,E2 -10931.59} C_VEL
LIN {X 0,Y 404.131,Z 224.145,A -85,B 0,C 180,E1 -10935.479,E2 -10935.479} C_VEL
LIN {X 0,Y 404.105,Z 224.144,A -85,B 0,C 180,E1 -10938.629,E2 -10938.629} C_VEL
LIN {X 0,Y 404.138,Z 224.144,A -85,B 0,C 180,E1 -10941.493,E2 -10941.493} C_VEL
LIN {X 0,Y 404.162,Z 224.137,A -85,B 0,C 180,E1 -10944.977,E2 -10944.977} C_VEL
LIN {X 0,Y 404.139,Z 224.143,A -85,B 0,C 180,E1 -10947.374,E2 -10947.374} C_VEL
LIN {X 0,Y 404.15,Z 224.138,A -85,B 0,C 180,E1 -10950.858,E2 -10950.858} C_VEL
LIN {X 0,Y 404.153,Z 224.138,A -85,B 0,C 180,E1 -10954.719,E2 -10954.719} C_VEL
LIN {X 0,Y 404.167,Z 224.142,A -85,B 0,C 180,E1 -10957.503,E2 -10957.503} C_VEL
LIN {X 0,Y 404.137,Z 224.14,A -85,B 0,C 180,E1 -10960.701,E2 -10960.701} C_VEL
LIN {X 0,Y 404.21,Z 224.135,A -85,B 0,C 180,E1 -10963.843,E2 -10963.843} C_VEL
LIN {X 0,Y 404.281,Z 224.123,A -85,B 0,C 180,E1 -10966.934,E2 -10966.934} C_VEL
LIN {X 0,Y 404.233,Z 224.13,A -85,B 0,C 180,E1 -10969.983,E2 -10969.983} C_VEL
LIN {X 0,Y 404.333,Z 224.117,A -85,B 0,C 180,E1 -10973.006,E2 -10973.006} C_VEL
LIN {X 0,Y 404.244,Z 224.128,A -85,B 0,C 180,E1 -10975.008,E2 -10975.008} C_VEL
LIN {X 0,Y 404.456,Z 224.102,A -85,B 0,C 180,E1 -10978.003,E2 -10978.003} C_VEL
LIN {X 0,Y 404.461,Z 224.101,A -85,B 0,C 180,E1 -10981.986,E2 -10981.986} C_VEL
LIN {X 0,Y 404.317,Z 224.117,A -85,B 0,C 180,E1 -10986.497,E2 -10986.497} C_VEL
LIN {X 0,Y 404.24,Z 224.129,A -85,B 0,C 180,E1 -10988.996,E2 -10988.996} C_VEL
LIN {X 0,Y 404.234,Z 224.129,A -85,B 0,C 180,E1 -10992.036,E2 -10992.036} C_VEL
LIN {X 0,Y 404.18,Z 224.138,A -85,B 0,C 180,E1 -10995.112,E2 -10995.112} C_VEL
LIN {X 0,Y 404.179,Z 224.135,A -85,B 0,C 180,E1 -10998.232,E2 -10998.232} C_VEL
LIN {X 0,Y 404.132,Z 224.148,A -85,B 0,C 180,E1 -11001.412,E2 -11001.412} C_VEL
LIN {X 0,Y 404.133,Z 224.141,A -85,B 0,C 180,E1 -11004.661,E2 -11004.661} C_VEL
LIN {X 0,Y 404.155,Z 224.139,A -85,B 0,C 180,E1 -11007.994,E2 -11007.994} C_VEL
LIN {X 0,Y 404.104,Z 224.149,A -85,B 0,C 180,E1 -11011.552,E2 -11011.552} C_VEL
LIN {X 0,Y 404.146,Z 224.142,A -85,B 0,C 180,E1 -11015.011,E2 -11015.011} C_VEL
LIN {X 0,Y 404.114,Z 224.144,A -85,B 0,C 180,E1 -11018.752,E2 -11018.752} C_VEL
LIN {X 0,Y 404.08,Z 224.151,A -85,B 0,C 180,E1 -11021.594,E2 -11021.594} C_VEL
LIN {X 0,Y 404.102,Z 224.145,A -85,B 0,C 180,E1 -11024.517,E2 -11024.517} C_VEL
LIN {X 0,Y 404.088,Z 224.153,A -85,B 0,C 180,E1 -11027.291,E2 -11027.291} C_VEL
LIN {X 0,Y 404.12,Z 224.142,A -85,B 0,C 180,E1 -11029.951,E2 -11029.951} C_VEL
LIN {X 0,Y 404.088,Z 224.152,A -85,B 0,C 180,E1 -11033.12,E2 -11033.12} C_VEL
LIN {X 0,Y 404.092,Z 224.145,A -85,B 0,C 180,E1 -11036.184,E2 -11036.184} C_VEL
LIN {X 0,Y 404.098,Z 224.146,A -85,B 0,C 180,E1 -11039.712,E2 -11039.712} C_VEL
LIN {X 0,Y 404.14,Z 224.146,A -85,B 0,C 180,E1 -11043.12,E2 -11043.12} C_VEL
LIN {X 0,Y 404.123,Z 224.142,A -85,B 0,C 180,E1 -11046.423,E2 -11046.423} C_VEL
LIN {X 0,Y 404.167,Z 224.137,A -85,B 0,C 180,E1 -11049.858,E2 -11049.858} C_VEL
LIN {X 0,Y 404.159,Z 224.143,A -85,B 0,C 180,E1 -11052.989,E2 -11052.989} C_VEL
LIN {X 0,Y 404.205,Z 224.135,A -85,B 0,C 180,E1 -11056.787,E2 -11056.787} C_VEL
LIN {X 0,Y 404.214,Z 224.13,A -85,B 0,C 180,E1 -11059.987,E2 -11059.987} C_VEL
LIN {X 0,Y 404.382,Z 224.116,A -85,B 0,C 180,E1 -11063.012,E2 -11063.012} C_VEL
LIN {X 0,Y 404.231,Z 224.135,A -85,B 0,C 180,E1 -11065.013,E2 -11065.013} C_VEL
LIN {X 0,Y 404.421,Z 224.104,A -85,B 0,C 180,E1 -11068.008,E2 -11068.008} C_VEL
LIN {X 0,Y 404.55,Z 224.088,A -85,B 0,C 180,E1 -11070,E2 -11070} C_VEL
LIN {X 0,Y 404.368,Z 224.118,A -85,B 0,C 180,E1 -11072.989,E2 -11072.989} C_VEL
LIN {X 0,Y 404.378,Z 224.117,A -85,B 0,C 180,E1 -11076.988,E2 -11076.988} C_VEL
LIN {X 0,Y 404.23,Z 224.225,A -85,B 0,C 180,E1 -11080.297,E2 -11080.297} C_VEL
LIN {X 0,Y 406.03,Z 234.113,A -85,B 0,C 180,E1 -11082.749,E2 -11082.749} C_VEL
LIN {X 0,Y 406.065,Z 237.218,A -85,B 0,C 180,E1 -11083.48,E2 -11083.48} C_VEL
LIN {X 0,Y 410.306,Z 259.089,A -85,B 0,C 180,E1 -11084.108,E2 -11084.108} C_VEL
LIN {X 0,Y 410.095,Z 271.776,A -85,B 0,C 180,E1 -11084.336,E2 -11084.336} C_VEL
LIN {X 0,Y 409.449,Z 277.618,A -85,B 0,C 180,E1 -11084.417,E2 -11084.417} C_VEL
LIN {X 0,Y 403.613,Z 296.595,A -85,B 0,C 180,E1 -11084.517,E2 -11084.517} C_VEL
LIN {X 0,Y 402.886,Z 302.443,A -85,B 0,C 180,E1 -11084.596,E2 -11084.596} C_VEL
LIN {X 0,Y 402.187,Z 345.757,A -85,B 0,C 180,E1 -11085.42,E2 -11085.42} C_VEL
LIN {X 0,Y 401.755,Z 359.094,A -85,B 0,C 180,E1 -11085.882,E2 -11085.882} C_VEL
LIN {X 0,Y 401.203,Z 371.825,A -85,B 0,C 180,E1 -11086.538,E2 -11086.538} C_VEL
LIN {X 0,Y 400.551,Z 383.521,A -85,B 0,C 180,E1 -11087.354,E2 -11087.354} C_VEL
LIN {X 0,Y 399.718,Z 395.729,A -85,B 0,C 180,E1 -11088.45,E2 -11088.45} C_VEL
LIN {X 0,Y 398.939,Z 405.481,A -85,B 0,C 180,E1 -11089.555,E2 -11089.555} C_VEL
LIN {X 0,Y 398.136,Z 415.187,A -85,B 0,C 180,E1 -11090.916,E2 -11090.916} C_VEL
LIN {X 0,Y 397.507,Z 423.413,A -85,B 0,C 180,E1 -11092.341,E2 -11092.341} C_VEL
LIN {X 0,Y 396.94,Z 430.124,A -85,B 0,C 180,E1 -11093.769,E2 -11093.769} C_VEL
LIN {X 0,Y 396.472,Z 435.992,A -85,B 0,C 180,E1 -11095.326,E2 -11095.326} C_VEL
LIN {X 0,Y 396.198,Z 440.6,A -85,B 0,C 180,E1 -11096.893,E2 -11096.893} C_VEL
LIN {X 0,Y 395.938,Z 444.392,A -85,B 0,C 180,E1 -11098.636,E2 -11098.636} C_VEL
LIN {X 0,Y 395.781,Z 446.251,A -85,B 0,C 180,E1 -11099.814,E2 -11099.814} C_VEL
LIN {X 0,Y 395.624,Z 447.934,A -85,B 0,C 180,E1 -11101.511,E2 -11101.511} C_VEL
LIN {X 0,Y 395.604,Z 448.464,A -85,B 0,C 180,E1 -11103.415,E2 -11103.415} C_VEL
LIN {X 0,Y 395.642,Z 447.699,A -85,B 0,C 180,E1 -11105.217,E2 -11105.217} C_VEL
LIN {X 0,Y 395.886,Z 445.529,A -85,B 0,C 180,E1 -11107.126,E2 -11107.126} C_VEL
LIN {X 0,Y 396.219,Z 441.585,A -85,B 0,C 180,E1 -11109.142,E2 -11109.142} C_VEL
LIN {X 0,Y 396.58,Z 436.46,A -85,B 0,C 180,E1 -11110.971,E2 -11110.971} C_VEL
LIN {X 0,Y 397.146,Z 430.47,A -85,B 0,C 180,E1 -11112.591,E2 -11112.591} C_VEL
LIN {X 0,Y 397.865,Z 422.657,A -85,B 0,C 180,E1 -11114.244,E2 -11114.244} C_VEL
LIN {X 0,Y 398.596,Z 414.498,A -85,B 0,C 180,E1 -11115.635,E2 -11115.635} C_VEL
LIN {X 0,Y 399.47,Z 405.176,A -85,B 0,C 180,E1 -11116.926,E2 -11116.926} C_VEL
LIN {X 0,Y 400.3,Z 394.881,A -85,B 0,C 180,E1 -11118.073,E2 -11118.073} C_VEL
LIN {X 0,Y 401.11,Z 383.911,A -85,B 0,C 180,E1 -11119.053,E2 -11119.053} C_VEL
LIN {X 0,Y 401.874,Z 372.203,A -85,B 0,C 180,E1 -11119.871,E2 -11119.871} C_VEL
LIN {X 0,Y 402.502,Z 359.286,A -85,B 0,C 180,E1 -11120.534,E2 -11120.534} C_VEL
LIN {X 0,Y 402.955,Z 346.563,A -85,B 0,C 180,E1 -11120.976,E2 -11120.976} C_VEL
LIN {X 0,Y 403.582,Z 307.788,A -85,B 0,C 180,E1 -11121.73,E2 -11121.73} C_VEL
LIN {X 0,Y 404.335,Z 259.356,A -85,B 0,C 180,E1 -11122.637,E2 -11122.637} C_VEL
LIN {X 0,Y 400.135,Z 239.711,A -85,B 0,C 180,E1 -11123.266,E2 -11123.266} C_VEL
LIN {X 0,Y 399.589,Z 237.674,A -85,B 0,C 180,E1 -11123.357,E2 -11123.357} C_VEL
LIN {X 0,Y 398.077,Z 229.434,A -85,B 0,C 180,E1 -11125.303,E2 -11125.303} C_VEL
LIN {X 0,Y 397.103,Z 225.023,A -85,B 0,C 180,E1 -11126.405,E2 -11126.405} C_VEL
LIN {X 0,Y 397.099,Z 225.023,A -85,B 0,C 180,E1 -11130.302,E2 -11130.302} C_VEL
LIN {X 0,Y 397.163,Z 225.013,A -85,B 0,C 180,E1 -11132.616,E2 -11132.616} C_VEL
LIN {X 0,Y 397.103,Z 225.018,A -85,B 0,C 180,E1 -11135.988,E2 -11135.988} C_VEL
LIN {X 0,Y 397.113,Z 225.018,A -85,B 0,C 180,E1 -11139.711,E2 -11139.711} C_VEL
LIN {X 0,Y 397.159,Z 225.014,A -85,B 0,C 180,E1 -11142.851,E2 -11142.851} C_VEL
LIN {X 0,Y 397.209,Z 225.009,A -85,B 0,C 180,E1 -11146.709,E2 -11146.709} C_VEL
LIN {X 0,Y 397.204,Z 225.006,A -85,B 0,C 180,E1 -11149.815,E2 -11149.815} C_VEL
LIN {X 0,Y 397.316,Z 224.997,A -85,B 0,C 180,E1 -11152.894,E2 -11152.894} C_VEL
LIN {X 0,Y 397.231,Z 225.002,A -85,B 0,C 180,E1 -11154.931,E2 -11154.931} C_VEL
LIN {X 0,Y 397.436,Z 224.974,A -85,B 0,C 180,E1 -11157.979,E2 -11157.979} C_VEL
LIN {X 0,Y 397.564,Z 224.96,A -85,B 0,C 180,E1 -11160.006,E2 -11160.006} C_VEL
LIN {X 0,Y 397.319,Z 224.993,A -85,B 0,C 180,E1 -11163.047,E2 -11163.047} C_VEL
LIN {X 0,Y 397.34,Z 224.983,A -85,B 0,C 180,E1 -11166.097,E2 -11166.097} C_VEL
LIN {X 0,Y 397.227,Z 224.999,A -85,B 0,C 180,E1 -11169.168,E2 -11169.168} C_VEL
LIN {X 0,Y 397.214,Z 225.006,A -85,B 0,C 180,E1 -11172.263,E2 -11172.263} C_VEL
LIN {X 0,Y 397.176,Z 225.008,A -85,B 0,C 180,E1 -11175.397,E2 -11175.397} C_VEL
LIN {X 0,Y 397.157,Z 225.009,A -85,B 0,C 180,E1 -11178.579,E2 -11178.579} C_VEL
LIN {X 0,Y 397.095,Z 225.017,A -85,B 0,C 180,E1 -11181.823,E2 -11181.823} C_VEL
LIN {X 0,Y 397.104,Z 225.016,A -85,B 0,C 180,E1 -11185.14,E2 -11185.14} C_VEL
LIN {X 0,Y 397.068,Z 225.026,A -85,B 0,C 180,E1 -11188.553,E2 -11188.553} C_VEL
LIN {X 0,Y 397.084,Z 225.021,A -85,B 0,C 180,E1 -11191.839,E2 -11191.839} C_VEL
LIN {X 0,Y 397.121,Z 225.018,A -85,B 0,C 180,E1 -11194.498,E2 -11194.498} C_VEL
LIN {X 0,Y 397.092,Z 225.023,A -85,B 0,C 180,E1 -11198.281,E2 -11198.281} C_VEL
LIN {X 0,Y 397.046,Z 225.03,A -85,B 0,C 180,E1 -11201.977,E2 -11201.977} C_VEL
LIN {X 0,Y 397.083,Z 225.024,A -85,B 0,C 180,E1 -11205.074,E2 -11205.074} C_VEL
LIN {X 0,Y 397.054,Z 225.026,A -85,B 0,C 180,E1 -11209.088,E2 -11209.088} C_VEL
LIN {X 0,Y 397.095,Z 225.021,A -85,B 0,C 180,E1 -11211.725,E2 -11211.725} C_VEL
LIN {X 0,Y 397.125,Z 225.017,A -85,B 0,C 180,E1 -11215.508,E2 -11215.508} C_VEL
LIN {X 0,Y 397.081,Z 225.027,A -85,B 0,C 180,E1 -11219.119,E2 -11219.119} C_VEL
LIN {X 0,Y 397.138,Z 225.103,A -85,B 0,C 180,E1 -11221.386,E2 -11221.386} C_VEL
LIN {X 0,Y 399.998,Z 238.78,A -85,B 0,C 180,E1 -11224.504,E2 -11224.504} C_VEL
LIN {X 0,Y 400.498,Z 243.774,A -85,B 0,C 180,E1 -11225.576,E2 -11225.576} C_VEL
LIN {X 0,Y 399.479,Z 257.368,A -85,B 0,C 180,E1 -11228.319,E2 -11228.319} C_VEL
LIN {X 0,Y 399.06,Z 264.26,A -85,B 0,C 180,E1 -11229.675,E2 -11229.675} C_VEL
LIN {X 0,Y 403.214,Z 289.324,A -85,B 0,C 180,E1 -11230.403,E2 -11230.403} C_VEL
LIN {X 0,Y 403.904,Z 295.579,A -85,B 0,C 180,E1 -11230.563,E2 -11230.563} C_VEL
LIN {X 0,Y 402.763,Z 372.955,A -85,B 0,C 180,E1 -11232.023,E2 -11232.023} C_VEL
LIN {X 0,Y 402.132,Z 386.062,A -85,B 0,C 180,E1 -11232.454,E2 -11232.454} C_VEL
LIN {X 0,Y 401.334,Z 398.745,A -85,B 0,C 180,E1 -11233.075,E2 -11233.075} C_VEL
LIN {X 0,Y 400.518,Z 410.072,A -85,B 0,C 180,E1 -11233.826,E2 -11233.826} C_VEL
LIN {X 0,Y 399.61,Z 421.78,A -85,B 0,C 180,E1 -11234.835,E2 -11234.835} C_VEL
LIN {X 0,Y 398.82,Z 431.861,A -85,B 0,C 180,E1 -11235.922,E2 -11235.922} C_VEL
LIN {X 0,Y 397.98,Z 441.847,A -85,B 0,C 180,E1 -11237.248,E2 -11237.248} C_VEL
LIN {X 0,Y 397.063,Z 451.025,A -85,B 0,C 180,E1 -11238.773,E2 -11238.773} C_VEL
LIN {X 0,Y 396.525,Z 458.439,A -85,B 0,C 180,E1 -11240.307,E2 -11240.307} C_VEL
LIN {X 0,Y 396.173,Z 464.396,A -85,B 0,C 180,E1 -11241.841,E2 -11241.841} C_VEL
LIN {X 0,Y 395.931,Z 469.1,A -85,B 0,C 180,E1 -11243.375,E2 -11243.375} C_VEL
LIN {X 0,Y 395.817,Z 472.692,A -85,B 0,C 180,E1 -11244.907,E2 -11244.907} C_VEL
LIN {X 0,Y 395.78,Z 474.519,A -85,B 0,C 180,E1 -11245.927,E2 -11245.927} C_VEL
LIN {X 0,Y 395.811,Z 476.893,A -85,B 0,C 180,E1 -11247.965,E2 -11247.965} C_VEL
LIN {X 0,Y 395.803,Z 477.485,A -85,B 0,C 180,E1 -11248.983,E2 -11248.983} C_VEL
LIN {X 0,Y 395.788,Z 477.644,A -85,B 0,C 180,E1 -11250,E2 -11250} C_VEL
LIN {X 0,Y 395.803,Z 477.393,A -85,B 0,C 180,E1 -11251.017,E2 -11251.017} C_VEL
LIN {X 0,Y 395.812,Z 476.75,A -85,B 0,C 180,E1 -11252.035,E2 -11252.035} C_VEL
LIN {X 0,Y 395.74,Z 475.708,A -85,B 0,C 180,E1 -11253.054,E2 -11253.054} C_VEL
LIN {X 0,Y 395.781,Z 474.218,A -85,B 0,C 180,E1 -11254.073,E2 -11254.073} C_VEL
LIN {X 0,Y 395.812,Z 470.781,A -85,B 0,C 180,E1 -11255.763,E2 -11255.763} C_VEL
LIN {X 0,Y 396.015,Z 467.057,A -85,B 0,C 180,E1 -11257.136,E2 -11257.136} C_VEL
LIN {X 0,Y 396.333,Z 460.735,A -85,B 0,C 180,E1 -11258.926,E2 -11258.926} C_VEL
LIN {X 0,Y 396.744,Z 453.843,A -85,B 0,C 180,E1 -11260.461,E2 -11260.461} C_VEL
LIN {X 0,Y 397.324,Z 446.811,A -85,B 0,C 180,E1 -11261.737,E2 -11261.737} C_VEL
LIN {X 0,Y 397.964,Z 438.335,A -85,B 0,C 180,E1 -11263.012,E2 -11263.012} C_VEL
LIN {X 0,Y 398.799,Z 427.865,A -85,B 0,C 180,E1 -11264.283,E2 -11264.283} C_VEL
LIN {X 0,Y 399.545,Z 417.505,A -85,B 0,C 180,E1 -11265.298,E2 -11265.298} C_VEL
LIN {X 0,Y 400.306,Z 406.163,A -85,B 0,C 180,E1 -11266.183,E2 -11266.183} C_VEL
LIN {X 0,Y 401.055,Z 394.625,A -85,B 0,C 180,E1 -11266.872,E2 -11266.872} C_VEL
LIN {X 0,Y 401.716,Z 381.423,A -85,B 0,C 180,E1 -11267.433,E2 -11267.433} C_VEL
LIN {X 0,Y 402.13,Z 368.757,A -85,B 0,C 180,E1 -11267.776,E2 -11267.776} C_VEL
LIN {X 0,Y 403.08,Z 293.49,A -85,B 0,C 180,E1 -11269.167,E2 -11269.167} C_VEL
LIN {X 0,Y 398.789,Z 265.072,A -85,B 0,C 180,E1 -11269.931,E2 -11269.931} C_VEL
LIN {X 0,Y 400.088,Z 247.347,A -85,B 0,C 180,E1 -11273.554,E2 -11273.554} C_VEL
LIN {X 0,Y 400.415,Z 241.992,A -85,B 0,C 180,E1 -11274.664,E2 -11274.664} C_VEL
LIN {X 0,Y 398.187,Z 230.186,A -85,B 0,C 180,E1 -11277.315,E2 -11277.315} C_VEL
LIN {X 0,Y 397.117,Z 225.021,A -85,B 0,C 180,E1 -11278.543,E2 -11278.543} C_VEL
LIN {X 0,Y 397.07,Z 225.024,A -85,B 0,C 180,E1 -11282.071,E2 -11282.071} C_VEL
LIN {X 0,Y 397.091,Z 225.021,A -85,B 0,C 180,E1 -11285.492,E2 -11285.492} C_VEL
LIN {X 0,Y 397.093,Z 225.017,A -85,B 0,C 180,E1 -11288.85,E2 -11288.85} C_VEL
LIN {X 0,Y 397.031,Z 225.027,A -85,B 0,C 180,E1 -11292.271,E2 -11292.271} C_VEL
LIN {X 0,Y 397.069,Z 225.021,A -85,B 0,C 180,E1 -11295.07,E2 -11295.07} C_VEL
LIN {X 0,Y 397.046,Z 225.027,A -85,B 0,C 180,E1 -11298.023,E2 -11298.023} C_VEL
LIN {X 0,Y 397.09,Z 225.025,A -85,B 0,C 180,E1 -11301.719,E2 -11301.719} C_VEL
LIN {X 0,Y 397.111,Z 225.02,A -85,B 0,C 180,E1 -11305.501,E2 -11305.501} C_VEL
LIN {X 0,Y 397.075,Z 225.021,A -85,B 0,C 180,E1 -11309.113,E2 -11309.113} C_VEL
LIN {X 0,Y 397.06,Z 225.023,A -85,B 0,C 180,E1 -11312.249,E2 -11312.249} C_VEL
LIN {X 0,Y 397.104,Z 225.016,A -85,B 0,C 180,E1 -11314.86,E2 -11314.86} C_VEL
LIN {X 0,Y 397.092,Z 225.019,A -85,B 0,C 180,E1 -11318.176,E2 -11318.176} C_VEL
LIN {X 0,Y 397.101,Z 225.021,A -85,B 0,C 180,E1 -11321.419,E2 -11321.419} C_VEL
LIN {X 0,Y 397.164,Z 225.008,A -85,B 0,C 180,E1 -11324.602,E2 -11324.602} C_VEL
LIN {X 0,Y 397.207,Z 225.008,A -85,B 0,C 180,E1 -11327.736,E2 -11327.736} C_VEL
LIN {X 0,Y 397.219,Z 225.002,A -85,B 0,C 180,E1 -11330.832,E2 -11330.832} C_VEL
LIN {X 0,Y 397.312,Z 224.993,A -85,B 0,C 180,E1 -11333.902,E2 -11333.902} C_VEL
LIN {X 0,Y 397.423,Z 224.978,A -85,B 0,C 180,E1 -11337.968,E2 -11337.968} C_VEL
LIN {X 0,Y 397.43,Z 224.977,A -85,B 0,C 180,E1 -11342.021,E2 -11342.021} C_VEL
LIN {X 0,Y 397.274,Z 224.995,A -85,B 0,C 180,E1 -11346.491,E2 -11346.491} C_VEL
LIN {X 0,Y 397.211,Z 225.006,A -85,B 0,C 180,E1 -11349.156,E2 -11349.156} C_VEL
LIN {X 0,Y 397.198,Z 225.005,A -85,B 0,C 180,E1 -11352.252,E2 -11352.252} C_VEL
LIN {X 0,Y 397.154,Z 225.016,A -85,B 0,C 180,E1 -11355.386,E2 -11355.386} C_VEL
LIN {X 0,Y 397.132,Z 225.013,A -85,B 0,C 180,E1 -11358.568,E2 -11358.568} C_VEL
LIN {X 0,Y 397.081,Z 225.021,A -85,B 0,C 180,E1 -11361.812,E2 -11361.812} C_VEL
LIN {X 0,Y 397.093,Z 225.021,A -85,B 0,C 180,E1 -11365.128,E2 -11365.128} C_VEL
LIN {X 0,Y 397.119,Z 225.017,A -85,B 0,C 180,E1 -11367.767,E2 -11367.767} C_VEL
LIN {X 0,Y 397.043,Z 225.026,A -85,B 0,C 180,E1 -11370.877,E2 -11370.877} C_VEL
LIN {X 0,Y 397.087,Z 225.018,A -85,B 0,C 180,E1 -11374.488,E2 -11374.488} C_VEL
LIN {X 0,Y 397.062,Z 225.021,A -85,B 0,C 180,E1 -11378.27,E2 -11378.27} C_VEL
LIN {X 0,Y 397.047,Z 225.026,A -85,B 0,C 180,E1 -11380.903,E2 -11380.903} C_VEL
LIN {X 0,Y 397.058,Z 225.025,A -85,B 0,C 180,E1 -11383.643,E2 -11383.643} C_VEL
LIN {X 0,Y 397.055,Z 225.022,A -85,B 0,C 180,E1 -11386.516,E2 -11386.516} C_VEL
LIN {X 0,Y 397.065,Z 225.021,A -85,B 0,C 180,E1 -11390.418,E2 -11390.418} C_VEL
LIN {X 0,Y 397.057,Z 225.022,A -85,B 0,C 180,E1 -11394.261,E2 -11394.261} C_VEL
LIN {X 0,Y 397.061,Z 225.023,A -85,B 0,C 180,E1 -11396.723,E2 -11396.723} C_VEL
LIN {X 0,Y 397.077,Z 225.019,A -85,B 0,C 180,E1 -11400.293,E2 -11400.293} C_VEL
LIN {X 0,Y 397.139,Z 225.013,A -85,B 0,C 180,E1 -11402.606,E2 -11402.606} C_VEL
LIN {X 0,Y 397.082,Z 225.019,A -85,B 0,C 180,E1 -11405.979,E2 -11405.979} C_VEL
LIN {X 0,Y 397.097,Z 225.023,A -85,B 0,C 180,E1 -11409.27,E2 -11409.27} C_VEL
LIN {X 0,Y 397.124,Z 225.017,A -85,B 0,C 180,E1 -11412.842,E2 -11412.842} C_VEL
LIN {X 0,Y 397.121,Z 225.015,A -85,B 0,C 180,E1 -11415.655,E2 -11415.655} C_VEL
LIN {X 0,Y 397.151,Z 225.013,A -85,B 0,C 180,E1 -11418.776,E2 -11418.776} C_VEL
LIN {X 0,Y 397.337,Z 224.987,A -85,B 0,C 180,E1 -11422.036,E2 -11422.036} C_VEL
LIN {X 0,Y 397.336,Z 224.987,A -85,B 0,C 180,E1 -11423.908,E2 -11423.908} C_VEL
LIN {X 0,Y 397.39,Z 224.98,A -85,B 0,C 180,E1 -11427.973,E2 -11427.973} C_VEL
LIN {X 0,Y 397.52,Z 224.964,A -85,B 0,C 180,E1 -11430,E2 -11430} C_VEL
LIN {X 0,Y 397.327,Z 224.995,A -85,B 0,C 180,E1 -11433.042,E2 -11433.042} C_VEL
LIN {X 0,Y 397.336,Z 224.988,A -85,B 0,C 180,E1 -11436.092,E2 -11436.092} C_VEL
LIN {X 0,Y 397.206,Z 225.009,A -85,B 0,C 180,E1 -11439.163,E2 -11439.163} C_VEL
LIN {X 0,Y 397.191,Z 225.109,A -85,B 0,C 180,E1 -11440.063,E2 -11440.063} C_VEL
LIN {X 0,Y 399.094,Z 235.634,A -85,B 0,C 180,E1 -11442.716,E2 -11442.716} C_VEL
LIN {X 0,Y 399.17,Z 237.511,A -85,B 0,C 180,E1 -11443.166,E2 -11443.166} C_VEL
LIN {X 0,Y 403.464,Z 259.055,A -85,B 0,C 180,E1 -11443.793,E2 -11443.793} C_VEL
LIN {X 0,Y 402.886,Z 302.443,A -85,B 0,C 180,E1 -11444.596,E2 -11444.596} C_VEL
LIN {X 0,Y 402.173,Z 308.282,A -85,B 0,C 180,E1 -11444.675,E2 -11444.675} C_VEL
LIN {X 0,Y 396.347,Z 327.244,A -85,B 0,C 180,E1 -11444.781,E2 -11444.781} C_VEL
LIN {X 0,Y 395.601,Z 333.085,A -85,B 0,C 180,E1 -11444.861,E2 -11444.861} C_VEL
LIN {X 0,Y 395.3,Z 349.475,A -85,B 0,C 180,E1 -11445.235,E2 -11445.235} C_VEL
LIN {X 0,Y 394.89,Z 361.051,A -85,B 0,C 180,E1 -11445.682,E2 -11445.682} C_VEL
LIN {X 0,Y 394.266,Z 373.854,A -85,B 0,C 180,E1 -11446.388,E2 -11446.388} C_VEL
LIN {X 0,Y 393.545,Z 385.838,A -85,B 0,C 180,E1 -11447.27,E2 -11447.27} C_VEL
LIN {X 0,Y 392.796,Z 396.263,A -85,B 0,C 180,E1 -11448.247,E2 -11448.247} C_VEL
LIN {X 0,Y 391.859,Z 407.05,A -85,B 0,C 180,E1 -11449.514,E2 -11449.514} C_VEL
LIN {X 0,Y 391.06,Z 416.376,A -85,B 0,C 180,E1 -11450.873,E2 -11450.873} C_VEL
LIN {X 0,Y 390.479,Z 423.837,A -85,B 0,C 180,E1 -11452.207,E2 -11452.207} C_VEL
LIN {X 0,Y 389.894,Z 430.449,A -85,B 0,C 180,E1 -11453.644,E2 -11453.644} C_VEL
LIN {X 0,Y 389.479,Z 435.588,A -85,B 0,C 180,E1 -11455.018,E2 -11455.018} C_VEL
LIN {X 0,Y 389.115,Z 440.941,A -85,B 0,C 180,E1 -11456.842,E2 -11456.842} C_VEL
LIN {X 0,Y 388.867,Z 444.71,A -85,B 0,C 180,E1 -11458.615,E2 -11458.615} C_VEL
LIN {X 0,Y 388.597,Z 447.253,A -85,B 0,C 180,E1 -11460.423,E2 -11460.423} C_VEL
LIN {X 0,Y 388.523,Z 448.339,A -85,B 0,C 180,E1 -11461.785,E2 -11461.785} C_VEL
LIN {X 0,Y 388.514,Z 448.693,A -85,B 0,C 180,E1 -11463.699,E2 -11463.699} C_VEL
LIN {X 0,Y 388.581,Z 447.77,A -85,B 0,C 180,E1 -11465.538,E2 -11465.538} C_VEL
LIN {X 0,Y 388.826,Z 445.642,A -85,B 0,C 180,E1 -11467.331,E2 -11467.331} C_VEL
LIN {X 0,Y 389.16,Z 442.027,A -85,B 0,C 180,E1 -11469.202,E2 -11469.202} C_VEL
LIN {X 0,Y 389.454,Z 437.977,A -85,B 0,C 180,E1 -11470.732,E2 -11470.732} C_VEL
LIN {X 0,Y 390.028,Z 432.306,A -85,B 0,C 180,E1 -11472.384,E2 -11472.384} C_VEL
LIN {X 0,Y 390.686,Z 425.325,A -85,B 0,C 180,E1 -11473.994,E2 -11473.994} C_VEL
LIN {X 0,Y 391.496,Z 416.69,A -85,B 0,C 180,E1 -11475.575,E2 -11475.575} C_VEL
LIN {X 0,Y 392.505,Z 406.564,A -85,B 0,C 180,E1 -11477.048,E2 -11477.048} C_VEL
LIN {X 0,Y 393.39,Z 396.427,A -85,B 0,C 180,E1 -11478.232,E2 -11478.232} C_VEL
LIN {X 0,Y 394.281,Z 385.388,A -85,B 0,C 180,E1 -11479.257,E2 -11479.257} C_VEL
LIN {X 0,Y 395.035,Z 374.138,A -85,B 0,C 180,E1 -11480.082,E2 -11480.082} C_VEL
LIN {X 0,Y 395.693,Z 361.839,A -85,B 0,C 180,E1 -11480.765,E2 -11480.765} C_VEL
LIN {X 0,Y 396.195,Z 348.799,A -85,B 0,C 180,E1 -11481.26,E2 -11481.26} C_VEL
LIN {X 0,Y 396.559,Z 331.157,A -85,B 0,C 180,E1 -11481.647,E2 -11481.647} C_VEL
LIN {X 0,Y 397.697,Z 260.031,A -85,B 0,C 180,E1 -11483.001,E2 -11483.001} C_VEL
LIN {X 0,Y 393.742,Z 241.811,A -85,B 0,C 180,E1 -11483.605,E2 -11483.605} C_VEL
LIN {X 0,Y 392.59,Z 237.999,A -85,B 0,C 180,E1 -11483.759,E2 -11483.759} C_VEL
LIN {X 0,Y 390.048,Z 225.903,A -85,B 0,C 180,E1 -11486.75,E2 -11486.75} C_VEL
LIN {X 0,Y 390.032,Z 225.903,A -85,B 0,C 180,E1 -11490.897,E2 -11490.897} C_VEL
LIN {X 0,Y 390.081,Z 225.893,A -85,B 0,C 180,E1 -11494.388,E2 -11494.388} C_VEL
LIN {X 0,Y 390.012,Z 225.901,A -85,B 0,C 180,E1 -11497.772,E2 -11497.772} C_VEL
LIN {X 0,Y 390.08,Z 225.9,A -85,B 0,C 180,E1 -11501.084,E2 -11501.084} C_VEL
LIN {X 0,Y 390.117,Z 225.892,A -85,B 0,C 180,E1 -11504.329,E2 -11504.329} C_VEL
LIN {X 0,Y 390.159,Z 225.883,A -85,B 0,C 180,E1 -11507.523,E2 -11507.523} C_VEL
LIN {X 0,Y 390.178,Z 225.883,A -85,B 0,C 180,E1 -11510.677,E2 -11510.677} C_VEL
LIN {X 0,Y 390.29,Z 225.866,A -85,B 0,C 180,E1 -11513.804,E2 -11513.804} C_VEL
LIN {X 0,Y 390.405,Z 225.85,A -85,B 0,C 180,E1 -11517.943,E2 -11517.943} C_VEL
LIN {X 0,Y 390.534,Z 225.836,A -85,B 0,C 180,E1 -11520.006,E2 -11520.006} C_VEL
LIN {X 0,Y 390.256,Z 225.873,A -85,B 0,C 180,E1 -11523.103,E2 -11523.103} C_VEL
LIN {X 0,Y 390.295,Z 225.861,A -85,B 0,C 180,E1 -11526.208,E2 -11526.208} C_VEL
LIN {X 0,Y 390.185,Z 225.875,A -85,B 0,C 180,E1 -11529.335,E2 -11529.335} C_VEL
LIN {X 0,Y 390.166,Z 225.886,A -85,B 0,C 180,E1 -11532.488,E2 -11532.488} C_VEL
LIN {X 0,Y 390.137,Z 225.885,A -85,B 0,C 180,E1 -11535.682,E2 -11535.682} C_VEL
LIN {X 0,Y 390.102,Z 225.889,A -85,B 0,C 180,E1 -11538.927,E2 -11538.927} C_VEL
LIN {X 0,Y 390.036,Z 225.896,A -85,B 0,C 180,E1 -11542.239,E2 -11542.239} C_VEL
LIN {X 0,Y 390.054,Z 225.893,A -85,B 0,C 180,E1 -11545.727,E2 -11545.727} C_VEL
LIN {X 0,Y 390.028,Z 225.897,A -85,B 0,C 180,E1 -11549.117,E2 -11549.117} C_VEL
LIN {X 0,Y 390.046,Z 225.896,A -85,B 0,C 180,E1 -11552.726,E2 -11552.726} C_VEL
LIN {X 0,Y 390.047,Z 225.898,A -85,B 0,C 180,E1 -11555.826,E2 -11555.826} C_VEL
LIN {X 0,Y 390.035,Z 225.897,A -85,B 0,C 180,E1 -11559.214,E2 -11559.214} C_VEL
LIN {X 0,Y 390.016,Z 225.905,A -85,B 0,C 180,E1 -11562.372,E2 -11562.372} C_VEL
LIN {X 0,Y 390.016,Z 225.904,A -85,B 0,C 180,E1 -11565.352,E2 -11565.352} C_VEL
LIN {X 0,Y 390.013,Z 225.909,A -85,B 0,C 180,E1 -11568.186,E2 -11568.186} C_VEL
LIN {X 0,Y 390.06,Z 225.897,A -85,B 0,C 180,E1 -11570.905,E2 -11570.905} C_VEL
LIN {X 0,Y 390.077,Z 225.897,A -85,B 0,C 180,E1 -11574.793,E2 -11574.793} C_VEL
LIN {X 0,Y 390.027,Z 225.907,A -85,B 0,C 180,E1 -11578.497,E2 -11578.497} C_VEL
LIN {X 0,Y 390.089,Z 225.941,A -85,B 0,C 180,E1 -11581.024,E2 -11581.024} C_VEL
LIN {X 0,Y 392.836,Z 238.897,A -85,B 0,C 180,E1 -11584.053,E2 -11584.053} C_VEL
LIN {X 0,Y 393.645,Z 243.997,A -85,B 0,C 180,E1 -11585.195,E2 -11585.195} C_VEL
LIN {X 0,Y 392.661,Z 257.243,A -85,B 0,C 180,E1 -11587.923,E2 -11587.923} C_VEL
LIN {X 0,Y 392.206,Z 263.783,A -85,B 0,C 180,E1 -11589.257,E2 -11589.257} C_VEL
LIN {X 0,Y 396.466,Z 289.04,A -85,B 0,C 180,E1 -11590.023,E2 -11590.023} C_VEL
LIN {X 0,Y 397.288,Z 296.859,A -85,B 0,C 180,E1 -11590.226,E2 -11590.226} C_VEL
LIN {X 0,Y 396.043,Z 373.458,A -85,B 0,C 180,E1 -11591.708,E2 -11591.708} C_VEL
LIN {X 0,Y 395.396,Z 386.287,A -85,B 0,C 180,E1 -11592.145,E2 -11592.145} C_VEL
LIN {X 0,Y 394.55,Z 398.829,A -85,B 0,C 180,E1 -11592.775,E2 -11592.775} C_VEL
LIN {X 0,Y 393.723,Z 410.056,A -85,B 0,C 180,E1 -11593.539,E2 -11593.539} C_VEL
LIN {X 0,Y 392.735,Z 421.712,A -85,B 0,C 180,E1 -11594.563,E2 -11594.563} C_VEL
LIN {X 0,Y 391.846,Z 432.561,A -85,B 0,C 180,E1 -11595.764,E2 -11595.764} C_VEL
LIN {X 0,Y 391.033,Z 441.712,A -85,B 0,C 180,E1 -11597.017,E2 -11597.017} C_VEL
LIN {X 0,Y 390.079,Z 450.867,A -85,B 0,C 180,E1 -11598.569,E2 -11598.569} C_VEL
LIN {X 0,Y 389.481,Z 458.264,A -85,B 0,C 180,E1 -11600.13,E2 -11600.13} C_VEL
LIN {X 0,Y 389.119,Z 464.206,A -85,B 0,C 180,E1 -11601.693,E2 -11601.693} C_VEL
LIN {X 0,Y 388.856,Z 468.895,A -85,B 0,C 180,E1 -11603.254,E2 -11603.254} C_VEL
LIN {X 0,Y 388.715,Z 472.471,A -85,B 0,C 180,E1 -11604.814,E2 -11604.814} C_VEL
LIN {X 0,Y 388.703,Z 474.285,A -85,B 0,C 180,E1 -11605.853,E2 -11605.853} C_VEL
LIN {X 0,Y 388.708,Z 476.645,A -85,B 0,C 180,E1 -11607.928,E2 -11607.928} C_VEL
LIN {X 0,Y 388.734,Z 477.232,A -85,B 0,C 180,E1 -11608.964,E2 -11608.964} C_VEL
LIN {X 0,Y 388.717,Z 477.379,A -85,B 0,C 180,E1 -11610,E2 -11610} C_VEL
LIN {X 0,Y 388.734,Z 477.122,A -85,B 0,C 180,E1 -11611.036,E2 -11611.036} C_VEL
LIN {X 0,Y 388.71,Z 476.471,A -85,B 0,C 180,E1 -11612.072,E2 -11612.072} C_VEL
LIN {X 0,Y 388.647,Z 475.422,A -85,B 0,C 180,E1 -11613.11,E2 -11613.11} C_VEL
LIN {X 0,Y 388.705,Z 473.92,A -85,B 0,C 180,E1 -11614.147,E2 -11614.147} C_VEL
LIN {X 0,Y 388.765,Z 469.881,A -85,B 0,C 180,E1 -11616.11,E2 -11616.11} C_VEL
LIN {X 0,Y 388.998,Z 465.089,A -85,B 0,C 180,E1 -11617.787,E2 -11617.787} C_VEL
LIN {X 0,Y 389.422,Z 458.236,A -85,B 0,C 180,E1 -11619.61,E2 -11619.61} C_VEL
LIN {X 0,Y 389.907,Z 450.769,A -85,B 0,C 180,E1 -11621.172,E2 -11621.172} C_VEL
LIN {X 0,Y 390.634,Z 443.167,A -85,B 0,C 180,E1 -11622.468,E2 -11622.468} C_VEL
LIN {X 0,Y 391.331,Z 434.572,A -85,B 0,C 180,E1 -11623.682,E2 -11623.682} C_VEL
LIN {X 0,Y 392.054,Z 424.973,A -85,B 0,C 180,E1 -11624.8,E2 -11624.8} C_VEL
LIN {X 0,Y 392.892,Z 413.929,A -85,B 0,C 180,E1 -11625.83,E2 -11625.83} C_VEL
LIN {X 0,Y 393.8,Z 401.569,A -85,B 0,C 180,E1 -11626.725,E2 -11626.725} C_VEL
LIN {X 0,Y 394.432,Z 389.879,A -85,B 0,C 180,E1 -11627.364,E2 -11627.364} C_VEL
LIN {X 0,Y 395.069,Z 377.455,A -85,B 0,C 180,E1 -11627.837,E2 -11627.837} C_VEL
LIN {X 0,Y 395.457,Z 360.174,A -85,B 0,C 180,E1 -11628.22,E2 -11628.22} C_VEL
LIN {X 0,Y 396.275,Z 293.93,A -85,B 0,C 180,E1 -11629.468,E2 -11629.468} C_VEL
LIN {X 0,Y 391.875,Z 264.864,A -85,B 0,C 180,E1 -11630.264,E2 -11630.264} C_VEL
LIN {X 0,Y 393.159,Z 248.263,A -85,B 0,C 180,E1 -11633.715,E2 -11633.715} C_VEL
LIN {X 0,Y 393.429,Z 243.042,A -85,B 0,C 180,E1 -11634.82,E2 -11634.82} C_VEL
LIN {X 0,Y 391.136,Z 231.099,A -85,B 0,C 180,E1 -11637.559,E2 -11637.559} C_VEL
LIN {X 0,Y 390.069,Z 225.899,A -85,B 0,C 180,E1 -11638.837,E2 -11638.837} C_VEL
LIN {X 0,Y 390.026,Z 225.898,A -85,B 0,C 180,E1 -11642.722,E2 -11642.722} C_VEL
LIN {X 0,Y 390.05,Z 225.895,A -85,B 0,C 180,E1 -11646.483,E2 -11646.483} C_VEL
LIN {X 0,Y 390.036,Z 225.898,A -85,B 0,C 180,E1 -11649.207,E2 -11649.207} C_VEL
LIN {X 0,Y 389.989,Z 225.903,A -85,B 0,C 180,E1 -11652.361,E2 -11652.361} C_VEL
LIN {X 0,Y 390.005,Z 225.903,A -85,B 0,C 180,E1 -11655.344,E2 -11655.344} C_VEL
LIN {X 0,Y 390.012,Z 225.902,A -85,B 0,C 180,E1 -11658.179,E2 -11658.179} C_VEL
LIN {X 0,Y 390.057,Z 225.894,A -85,B 0,C 180,E1 -11660.899,E2 -11660.899} C_VEL
LIN {X 0,Y 390.065,Z 225.893,A -85,B 0,C 180,E1 -11664.786,E2 -11664.786} C_VEL
LIN {X 0,Y 390.03,Z 225.902,A -85,B 0,C 180,E1 -11667.874,E2 -11667.874} C_VEL
LIN {X 0,Y 390.025,Z 225.898,A -85,B 0,C 180,E1 -11670.883,E2 -11670.883} C_VEL
LIN {X 0,Y 390.065,Z 225.893,A -85,B 0,C 180,E1 -11674.374,E2 -11674.374} C_VEL
LIN {X 0,Y 390.035,Z 225.902,A -85,B 0,C 180,E1 -11677.761,E2 -11677.761} C_VEL
LIN {X 0,Y 390.053,Z 225.896,A -85,B 0,C 180,E1 -11681.07,E2 -11681.07} C_VEL
LIN {X 0,Y 390.127,Z 225.886,A -85,B 0,C 180,E1 -11684.318,E2 -11684.318} C_VEL
LIN {X 0,Y 390.162,Z 225.887,A -85,B 0,C 180,E1 -11687.511,E2 -11687.511} C_VEL
LIN {X 0,Y 390.178,Z 225.879,A -85,B 0,C 180,E1 -11690.665,E2 -11690.665} C_VEL
LIN {X 0,Y 390.267,Z 225.872,A -85,B 0,C 180,E1 -11693.792,E2 -11693.792} C_VEL
LIN {X 0,Y 390.39,Z 225.855,A -85,B 0,C 180,E1 -11697.931,E2 -11697.931} C_VEL
LIN {X 0,Y 390.397,Z 225.853,A -85,B 0,C 180,E1 -11702.057,E2 -11702.057} C_VEL
LIN {X 0,Y 390.235,Z 225.872,A -85,B 0,C 180,E1 -11706.483,E2 -11706.483} C_VEL
LIN {X 0,Y 390.17,Z 225.885,A -85,B 0,C 180,E1 -11709.323,E2 -11709.323} C_VEL
LIN {X 0,Y 390.15,Z 225.882,A -85,B 0,C 180,E1 -11712.477,E2 -11712.477} C_VEL
LIN {X 0,Y 390.115,Z 225.891,A -85,B 0,C 180,E1 -11715.671,E2 -11715.671} C_VEL
LIN {X 0,Y 390.077,Z 225.893,A -85,B 0,C 180,E1 -11718.916,E2 -11718.916} C_VEL
LIN {X 0,Y 390.018,Z 225.899,A -85,B 0,C 180,E1 -11722.228,E2 -11722.228} C_VEL
LIN {X 0,Y 390.055,Z 225.897,A -85,B 0,C 180,E1 -11725.727,E2 -11725.727} C_VEL
LIN {X 0,Y 390.058,Z 225.895,A -85,B 0,C 180,E1 -11728.012,E2 -11728.012} C_VEL
LIN {X 0,Y 389.988,Z 225.908,A -85,B 0,C 180,E1 -11731.499,E2 -11731.499} C_VEL
LIN {X 0,Y 390.046,Z 225.901,A -85,B 0,C 180,E1 -11735.201,E2 -11735.201} C_VEL
LIN {X 0,Y 390.029,Z 225.903,A -85,B 0,C 180,E1 -11739.213,E2 -11739.213} C_VEL
LIN {X 0,Y 390,Z 225.901,A -85,B 0,C 180,E1 -11742.369,E2 -11742.369} C_VEL
LIN {X 0,Y 389.999,Z 225.907,A -85,B 0,C 180,E1 -11745.349,E2 -11745.349} C_VEL
LIN {X 0,Y 389.982,Z 225.903,A -85,B 0,C 180,E1 -11748.182,E2 -11748.182} C_VEL
LIN {X 0,Y 390.041,Z 225.899,A -85,B 0,C 180,E1 -11750.903,E2 -11750.903} C_VEL
LIN {X 0,Y 390.033,Z 225.899,A -85,B 0,C 180,E1 -11754.789,E2 -11754.789} C_VEL
LIN {X 0,Y 389.972,Z 225.905,A -85,B 0,C 180,E1 -11758.492,E2 -11758.492} C_VEL
LIN {X 0,Y 390.062,Z 225.893,A -85,B 0,C 180,E1 -11762.066,E2 -11762.066} C_VEL
LIN {X 0,Y 390.027,Z 225.901,A -85,B 0,C 180,E1 -11765.516,E2 -11765.516} C_VEL
LIN {X 0,Y 390.047,Z 225.899,A -85,B 0,C 180,E1 -11768.878,E2 -11768.878} C_VEL
LIN {X 0,Y 390.09,Z 225.892,A -85,B 0,C 180,E1 -11772.689,E2 -11772.689} C_VEL
LIN {X 0,Y 390.134,Z 225.886,A -85,B 0,C 180,E1 -11776.56,E2 -11776.56} C_VEL
LIN {X 0,Y 390.12,Z 225.888,A -85,B 0,C 180,E1 -11779.622,E2 -11779.622} C_VEL
LIN {X 0,Y 390.281,Z 225.869,A -85,B 0,C 180,E1 -11782.759,E2 -11782.759} C_VEL
LIN {X 0,Y 390.175,Z 225.883,A -85,B 0,C 180,E1 -11784.833,E2 -11784.833} C_VEL
LIN {X 0,Y 390.359,Z 225.856,A -85,B 0,C 180,E1 -11787.936,E2 -11787.936} C_VEL
LIN {X 0,Y 390.489,Z 225.84,A -85,B 0,C 180,E1 -11790,E2 -11790} C_VEL
LIN {X 0,Y 390.286,Z 225.871,A -85,B 0,C 180,E1 -11793.097,E2 -11793.097} C_VEL
LIN {X 0,Y 390.289,Z 225.866,A -85,B 0,C 180,E1 -11796.202,E2 -11796.202} C_VEL
LIN {X 0,Y 390.16,Z 225.887,A -85,B 0,C 180,E1 -11799.33,E2 -11799.33} C_VEL
LIN {X 0,Y 390.177,Z 226.105,A -85,B 0,C 180,E1 -11799.852,E2 -11799.852} C_VEL
LIN {X 0,Y 392.048,Z 236.132,A -85,B 0,C 180,E1 -11802.422,E2 -11802.422} C_VEL
LIN {X 0,Y 392.201,Z 237.701,A -85,B 0,C 180,E1 -11802.812,E2 -11802.812} C_VEL
LIN {X 0,Y 396.801,Z 260.482,A -85,B 0,C 180,E1 -11803.507,E2 -11803.507} C_VEL
LIN {X 0,Y 395.601,Z 333.085,A -85,B 0,C 180,E1 -11804.861,E2 -11804.861} C_VEL
LIN {X 0,Y 394.845,Z 338.918,A -85,B 0,C 180,E1 -11804.941,E2 -11804.941} C_VEL
LIN {X 0,Y 391.917,Z 348.361,A -85,B 0,C 180,E1 -11805.054,E2 -11805.054} C_VEL
LIN {X 0,Y 388.894,Z 357.668,A -85,B 0,C 180,E1 -11805.266,E2 -11805.266} C_VEL
LIN {X 0,Y 387.958,Z 363.282,A -85,B 0,C 180,E1 -11805.495,E2 -11805.495} C_VEL
LIN {X 0,Y 387.293,Z 376.502,A -85,B 0,C 180,E1 -11806.274,E2 -11806.274} C_VEL
LIN {X 0,Y 386.527,Z 388.055,A -85,B 0,C 180,E1 -11807.185,E2 -11807.185} C_VEL
LIN {X 0,Y 385.604,Z 399.855,A -85,B 0,C 180,E1 -11808.376,E2 -11808.376} C_VEL
LIN {X 0,Y 384.713,Z 409.662,A -85,B 0,C 180,E1 -11809.613,E2 -11809.613} C_VEL
LIN {X 0,Y 383.938,Z 418.683,A -85,B 0,C 180,E1 -11811.029,E2 -11811.029} C_VEL
LIN {X 0,Y 383.152,Z 427.05,A -85,B 0,C 180,E1 -11812.655,E2 -11812.655} C_VEL
LIN {X 0,Y 382.598,Z 434.172,A -85,B 0,C 180,E1 -11814.412,E2 -11814.412} C_VEL
LIN {X 0,Y 382.133,Z 439.733,A -85,B 0,C 180,E1 -11816.192,E2 -11816.192} C_VEL
LIN {X 0,Y 381.918,Z 443.899,A -85,B 0,C 180,E1 -11817.978,E2 -11817.978} C_VEL
LIN {X 0,Y 381.558,Z 447.139,A -85,B 0,C 180,E1 -11820.055,E2 -11820.055} C_VEL
LIN {X 0,Y 381.415,Z 448.733,A -85,B 0,C 180,E1 -11822.065,E2 -11822.065} C_VEL
LIN {X 0,Y 381.404,Z 448.924,A -85,B 0,C 180,E1 -11823.999,E2 -11823.999} C_VEL
LIN {X 0,Y 381.56,Z 447.553,A -85,B 0,C 180,E1 -11826.114,E2 -11826.114} C_VEL
LIN {X 0,Y 381.801,Z 445.493,A -85,B 0,C 180,E1 -11827.686,E2 -11827.686} C_VEL
LIN {X 0,Y 382.122,Z 442.067,A -85,B 0,C 180,E1 -11829.438,E2 -11829.438} C_VEL
LIN {X 0,Y 382.482,Z 437.54,A -85,B 0,C 180,E1 -11831.13,E2 -11831.13} C_VEL
LIN {X 0,Y 383.106,Z 431.712,A -85,B 0,C 180,E1 -11832.807,E2 -11832.807} C_VEL
LIN {X 0,Y 383.863,Z 424.482,A -85,B 0,C 180,E1 -11834.448,E2 -11834.448} C_VEL
LIN {X 0,Y 384.747,Z 415.576,A -85,B 0,C 180,E1 -11836.054,E2 -11836.054} C_VEL
LIN {X 0,Y 385.751,Z 405.897,A -85,B 0,C 180,E1 -11837.455,E2 -11837.455} C_VEL
LIN {X 0,Y 386.617,Z 396.298,A -85,B 0,C 180,E1 -11838.576,E2 -11838.576} C_VEL
LIN {X 0,Y 387.63,Z 384.251,A -85,B 0,C 180,E1 -11839.694,E2 -11839.694} C_VEL
LIN {X 0,Y 388.427,Z 372.784,A -85,B 0,C 180,E1 -11840.522,E2 -11840.522} C_VEL
LIN {X 0,Y 389.123,Z 359.856,A -85,B 0,C 180,E1 -11841.208,E2 -11841.208} C_VEL
LIN {X 0,Y 389.604,Z 346.405,A -85,B 0,C 180,E1 -11841.69,E2 -11841.69} C_VEL
LIN {X 0,Y 391.137,Z 261.224,A -85,B 0,C 180,E1 -11843.363,E2 -11843.363} C_VEL
LIN {X 0,Y 387.135,Z 242.961,A -85,B 0,C 180,E1 -11843.99,E2 -11843.99} C_VEL
LIN {X 0,Y 385.51,Z 238.282,A -85,B 0,C 180,E1 -11844.205,E2 -11844.205} C_VEL
LIN {X 0,Y 382.985,Z 226.782,A -85,B 0,C 180,E1 -11847.112,E2 -11847.112} C_VEL
LIN {X 0,Y 382.964,Z 226.784,A -85,B 0,C 180,E1 -11850.307,E2 -11850.307} C_VEL
LIN {X 0,Y 383.025,Z 226.774,A -85,B 0,C 180,E1 -11852.704,E2 -11852.704} C_VEL
LIN {X 0,Y 383.022,Z 226.777,A -85,B 0,C 180,E1 -11855.046,E2 -11855.046} C_VEL
LIN {X 0,Y 382.966,Z 226.781,A -85,B 0,C 180,E1 -11858.475,E2 -11858.475} C_VEL
LIN {X 0,Y 383.039,Z 226.773,A -85,B 0,C 180,E1 -11861.833,E2 -11861.833} C_VEL
LIN {X 0,Y 383.09,Z 226.765,A -85,B 0,C 180,E1 -11865.125,E2 -11865.125} C_VEL
LIN {X 0,Y 383.088,Z 226.763,A -85,B 0,C 180,E1 -11868.364,E2 -11868.364} C_VEL
LIN {X 0,Y 383.211,Z 226.745,A -85,B 0,C 180,E1 -11872.021,E2 -11872.021} C_VEL
LIN {X 0,Y 383.174,Z 226.752,A -85,B 0,C 180,E1 -11874.744,E2 -11874.744} C_VEL
LIN {X 0,Y 383.372,Z 226.726,A -85,B 0,C 180,E1 -11877.905,E2 -11877.905} C_VEL
LIN {X 0,Y 383.503,Z 226.712,A -85,B 0,C 180,E1 -11880.006,E2 -11880.006} C_VEL
LIN {X 0,Y 383.194,Z 226.752,A -85,B 0,C 180,E1 -11883.16,E2 -11883.16} C_VEL
LIN {X 0,Y 383.252,Z 226.738,A -85,B 0,C 180,E1 -11886.322,E2 -11886.322} C_VEL
LIN {X 0,Y 383.135,Z 226.752,A -85,B 0,C 180,E1 -11889.508,E2 -11889.508} C_VEL
LIN {X 0,Y 383.124,Z 226.755,A -85,B 0,C 180,E1 -11893.541,E2 -11893.541} C_VEL
LIN {X 0,Y 383.094,Z 226.762,A -85,B 0,C 180,E1 -11897.074,E2 -11897.074} C_VEL
LIN {X 0,Y 383.03,Z 226.775,A -85,B 0,C 180,E1 -11900.651,E2 -11900.651} C_VEL
LIN {X 0,Y 383.01,Z 226.771,A -85,B 0,C 180,E1 -11903.814,E2 -11903.814} C_VEL
LIN {X 0,Y 382.971,Z 226.776,A -85,B 0,C 180,E1 -11907.313,E2 -11907.313} C_VEL
LIN {X 0,Y 382.985,Z 226.778,A -85,B 0,C 180,E1 -11910.923,E2 -11910.923} C_VEL
LIN {X 0,Y 383.017,Z 226.776,A -85,B 0,C 180,E1 -11914.673,E2 -11914.673} C_VEL
LIN {X 0,Y 382.997,Z 226.776,A -85,B 0,C 180,E1 -11917.905,E2 -11917.905} C_VEL
LIN {X 0,Y 382.964,Z 226.781,A -85,B 0,C 180,E1 -11921.355,E2 -11921.355} C_VEL
LIN {X 0,Y 382.973,Z 226.785,A -85,B 0,C 180,E1 -11924.302,E2 -11924.302} C_VEL
LIN {X 0,Y 382.986,Z 226.779,A -85,B 0,C 180,E1 -11927.238,E2 -11927.238} C_VEL
LIN {X 0,Y 382.99,Z 226.781,A -85,B 0,C 180,E1 -11930.423,E2 -11930.423} C_VEL
LIN {X 0,Y 383.022,Z 226.776,A -85,B 0,C 180,E1 -11934.045,E2 -11934.045} C_VEL
LIN {X 0,Y 383.01,Z 226.777,A -85,B 0,C 180,E1 -11936.601,E2 -11936.601} C_VEL
LIN {X 0,Y 383.004,Z 226.782,A -85,B 0,C 180,E1 -11940.302,E2 -11940.302} C_VEL
LIN {X 0,Y 383.04,Z 226.94,A -85,B 0,C 180,E1 -11940.683,E2 -11940.683} C_VEL
LIN {X 0,Y 385.871,Z 239.994,A -85,B 0,C 180,E1 -11943.81,E2 -11943.81} C_VEL
LIN {X 0,Y 386.729,Z 245.228,A -85,B 0,C 180,E1 -11945.007,E2 -11945.007} C_VEL
LIN {X 0,Y 385.86,Z 257.139,A -85,B 0,C 180,E1 -11947.513,E2 -11947.513} C_VEL
LIN {X 0,Y 385.404,Z 263.75,A -85,B 0,C 180,E1 -11948.847,E2 -11948.847} C_VEL
LIN {X 0,Y 389.654,Z 288.367,A -85,B 0,C 180,E1 -11949.617,E2 -11949.617} C_VEL
LIN {X 0,Y 390.687,Z 296.996,A -85,B 0,C 180,E1 -11949.853,E2 -11949.853} C_VEL
LIN {X 0,Y 389.385,Z 373.047,A -85,B 0,C 180,E1 -11951.349,E2 -11951.349} C_VEL
LIN {X 0,Y 388.71,Z 385.914,A -85,B 0,C 180,E1 -11951.794,E2 -11951.794} C_VEL
LIN {X 0,Y 387.792,Z 399.018,A -85,B 0,C 180,E1 -11952.465,E2 -11952.465} C_VEL
LIN {X 0,Y 386.93,Z 410.103,A -85,B 0,C 180,E1 -11953.242,E2 -11953.242} C_VEL
LIN {X 0,Y 385.901,Z 421.686,A -85,B 0,C 180,E1 -11954.283,E2 -11954.283} C_VEL
LIN {X 0,Y 384.932,Z 432.478,A -85,B 0,C 180,E1 -11955.503,E2 -11955.503} C_VEL
LIN {X 0,Y 384.092,Z 441.576,A -85,B 0,C 180,E1 -11956.779,E2 -11956.779} C_VEL
LIN {X 0,Y 383.109,Z 450.71,A -85,B 0,C 180,E1 -11958.359,E2 -11958.359} C_VEL
LIN {X 0,Y 382.462,Z 458.089,A -85,B 0,C 180,E1 -11959.947,E2 -11959.947} C_VEL
LIN {X 0,Y 382.054,Z 464.015,A -85,B 0,C 180,E1 -11961.538,E2 -11961.538} C_VEL
LIN {X 0,Y 381.773,Z 468.688,A -85,B 0,C 180,E1 -11963.128,E2 -11963.128} C_VEL
LIN {X 0,Y 381.621,Z 472.252,A -85,B 0,C 180,E1 -11964.717,E2 -11964.717} C_VEL
LIN {X 0,Y 381.626,Z 474.053,A -85,B 0,C 180,E1 -11965.776,E2 -11965.776} C_VEL
LIN {X 0,Y 381.606,Z 476.399,A -85,B 0,C 180,E1 -11967.889,E2 -11967.889} C_VEL
LIN {X 0,Y 381.648,Z 476.978,A -85,B 0,C 180,E1 -11968.945,E2 -11968.945} C_VEL
LIN {X 0,Y 381.649,Z 477.113,A -85,B 0,C 180,E1 -11970,E2 -11970} C_VEL
LIN {X 0,Y 381.648,Z 476.848,A -85,B 0,C 180,E1 -11971.055,E2 -11971.055} C_VEL
LIN {X 0,Y 381.609,Z 476.189,A -85,B 0,C 180,E1 -11972.111,E2 -11972.111} C_VEL
LIN {X 0,Y 381.558,Z 475.129,A -85,B 0,C 180,E1 -11973.168,E2 -11973.168} C_VEL
LIN {X 0,Y 381.629,Z 473.612,A -85,B 0,C 180,E1 -11974.224,E2 -11974.224} C_VEL
LIN {X 0,Y 381.692,Z 469.841,A -85,B 0,C 180,E1 -11976.103,E2 -11976.103} C_VEL
LIN {X 0,Y 381.92,Z 464.739,A -85,B 0,C 180,E1 -11977.933,E2 -11977.933} C_VEL
LIN {X 0,Y 382.371,Z 457.85,A -85,B 0,C 180,E1 -11979.789,E2 -11979.789} C_VEL
LIN {X 0,Y 382.91,Z 450.356,A -85,B 0,C 180,E1 -11981.379,E2 -11981.379} C_VEL
LIN {X 0,Y 383.646,Z 442.721,A -85,B 0,C 180,E1 -11982.699,E2 -11982.699} C_VEL
LIN {X 0,Y 384.45,Z 433.595,A -85,B 0,C 180,E1 -11983.999,E2 -11983.999} C_VEL
LIN {X 0,Y 385.209,Z 423.141,A -85,B 0,C 180,E1 -11985.204,E2 -11985.204} C_VEL
LIN {X 0,Y 386.145,Z 411.714,A -85,B 0,C 180,E1 -11986.25,E2 -11986.25} C_VEL
LIN {X 0,Y 387.012,Z 399.846,A -85,B 0,C 180,E1 -11987.095,E2 -11987.095} C_VEL
LIN {X 0,Y 387.802,Z 386.761,A -85,B 0,C 180,E1 -11987.773,E2 -11987.773} C_VEL
LIN {X 0,Y 388.405,Z 373.928,A -85,B 0,C 180,E1 -11988.221,E2 -11988.221} C_VEL
LIN {X 0,Y 389.596,Z 295.332,A -85,B 0,C 180,E1 -11989.754,E2 -11989.754} C_VEL
LIN {X 0,Y 384.976,Z 264.568,A -85,B 0,C 180,E1 -11990.622,E2 -11990.622} C_VEL
LIN {X 0,Y 386.32,Z 248.056,A -85,B 0,C 180,E1 -11994.123,E2 -11994.123} C_VEL
LIN {X 0,Y 386.441,Z 243.954,A -85,B 0,C 180,E1 -11995.013,E2 -11995.013} C_VEL
LIN {X 0,Y 383.735,Z 230.203,A -85,B 0,C 180,E1 -11998.239,E2 -11998.239} C_VEL
LIN {X 0,Y 383.017,Z 226.777,A -85,B 0,C 180,E1 -11999.094,E2 -11999.094} C_VEL
LIN {X 0,Y 382.974,Z 226.777,A -85,B 0,C 180,E1 -12002.413,E2 -12002.413} C_VEL
LIN {X 0,Y 383.021,Z 226.773,A -85,B 0,C 180,E1 -12006.157,E2 -12006.157} C_VEL
LIN {X 0,Y 382.989,Z 226.779,A -85,B 0,C 180,E1 -12009.577,E2 -12009.577} C_VEL
LIN {X 0,Y 382.94,Z 226.78,A -85,B 0,C 180,E1 -12012.768,E2 -12012.768} C_VEL
LIN {X 0,Y 382.946,Z 226.786,A -85,B 0,C 180,E1 -12015.777,E2 -12015.777} C_VEL
LIN {X 0,Y 382.967,Z 226.777,A -85,B 0,C 180,E1 -12018.798,E2 -12018.798} C_VEL
LIN {X 0,Y 382.995,Z 226.776,A -85,B 0,C 180,E1 -12022.095,E2 -12022.095} C_VEL
LIN {X 0,Y 383.021,Z 226.777,A -85,B 0,C 180,E1 -12025.657,E2 -12025.657} C_VEL
LIN {X 0,Y 382.982,Z 226.776,A -85,B 0,C 180,E1 -12029.077,E2 -12029.077} C_VEL
LIN {X 0,Y 382.968,Z 226.777,A -85,B 0,C 180,E1 -12032.686,E2 -12032.686} C_VEL
LIN {X 0,Y 383.01,Z 226.773,A -85,B 0,C 180,E1 -12036.186,E2 -12036.186} C_VEL
LIN {X 0,Y 383.038,Z 226.775,A -85,B 0,C 180,E1 -12039.592,E2 -12039.592} C_VEL
LIN {X 0,Y 383.077,Z 226.764,A -85,B 0,C 180,E1 -12042.925,E2 -12042.925} C_VEL
LIN {X 0,Y 383.124,Z 226.758,A -85,B 0,C 180,E1 -12046.459,E2 -12046.459} C_VEL
LIN {X 0,Y 383.129,Z 226.757,A -85,B 0,C 180,E1 -12050.492,E2 -12050.492} C_VEL
LIN {X 0,Y 383.226,Z 226.75,A -85,B 0,C 180,E1 -12053.677,E2 -12053.677} C_VEL
LIN {X 0,Y 383.355,Z 226.732,A -85,B 0,C 180,E1 -12057.893,E2 -12057.893} C_VEL
LIN {X 0,Y 383.363,Z 226.729,A -85,B 0,C 180,E1 -12062.095,E2 -12062.095} C_VEL
LIN {X 0,Y 383.2,Z 226.748,A -85,B 0,C 180,E1 -12066.471,E2 -12066.471} C_VEL
LIN {X 0,Y 383.121,Z 226.765,A -85,B 0,C 180,E1 -12069.496,E2 -12069.496} C_VEL
LIN {X 0,Y 383.106,Z 226.766,A -85,B 0,C 180,E1 -12073.53,E2 -12073.53} C_VEL
LIN {X 0,Y 383.071,Z 226.767,A -85,B 0,C 180,E1 -12077.063,E2 -12077.063} C_VEL
LIN {X 0,Y 383.005,Z 226.773,A -85,B 0,C 180,E1 -12080.641,E2 -12080.641} C_VEL
LIN {X 0,Y 382.989,Z 226.777,A -85,B 0,C 180,E1 -12083.802,E2 -12083.802} C_VEL
LIN {X 0,Y 383.017,Z 226.777,A -85,B 0,C 180,E1 -12087.297,E2 -12087.297} C_VEL
LIN {X 0,Y 382.948,Z 226.782,A -85,B 0,C 180,E1 -12090.913,E2 -12090.913} C_VEL
LIN {X 0,Y 382.981,Z 226.776,A -85,B 0,C 180,E1 -12094.662,E2 -12094.662} C_VEL
LIN {X 0,Y 382.959,Z 226.779,A -85,B 0,C 180,E1 -12097.898,E2 -12097.898} C_VEL
LIN {X 0,Y 382.942,Z 226.787,A -85,B 0,C 180,E1 -12101.342,E2 -12101.342} C_VEL
LIN {X 0,Y 382.952,Z 226.779,A -85,B 0,C 180,E1 -12104.298,E2 -12104.298} C_VEL
LIN {X 0,Y 382.964,Z 226.784,A -85,B 0,C 180,E1 -12107.235,E2 -12107.235} C_VEL
LIN {X 0,Y 382.966,Z 226.777,A -85,B 0,C 180,E1 -12110.409,E2 -12110.409} C_VEL
LIN {X 0,Y 382.975,Z 226.776,A -85,B 0,C 180,E1 -12114.04,E2 -12114.04} C_VEL
LIN {X 0,Y 382.934,Z 226.784,A -85,B 0,C 180,E1 -12117.574,E2 -12117.574} C_VEL
LIN {X 0,Y 382.942,Z 226.78,A -85,B 0,C 180,E1 -12120.297,E2 -12120.297} C_VEL
LIN {X 0,Y 383.001,Z 226.775,A -85,B 0,C 180,E1 -12122.695,E2 -12122.695} C_VEL
LIN {X 0,Y 382.99,Z 226.774,A -85,B 0,C 180,E1 -12126.19,E2 -12126.19} C_VEL
LIN {X 0,Y 383.023,Z 226.772,A -85,B 0,C 180,E1 -12129.597,E2 -12129.597} C_VEL
LIN {X 0,Y 383.047,Z 226.772,A -85,B 0,C 180,E1 -12132.929,E2 -12132.929} C_VEL
LIN {X 0,Y 383.066,Z 226.766,A -85,B 0,C 180,E1 -12136.462,E2 -12136.462} C_VEL
LIN {X 0,Y 383.082,Z 226.766,A -85,B 0,C 180,E1 -12139.429,E2 -12139.429} C_VEL
LIN {X 0,Y 383.232,Z 226.746,A -85,B 0,C 180,E1 -12142.625,E2 -12142.625} C_VEL
LIN {X 0,Y 383.148,Z 226.758,A -85,B 0,C 180,E1 -12144.738,E2 -12144.738} C_VEL
LIN {X 0,Y 383.328,Z 226.732,A -85,B 0,C 180,E1 -12147.899,E2 -12147.899} C_VEL
LIN {X 0,Y 383.459,Z 226.716,A -85,B 0,C 180,E1 -12150,E2 -12150} C_VEL
LIN {X 0,Y 383.221,Z 226.751,A -85,B 0,C 180,E1 -12153.154,E2 -12153.154} C_VEL
LIN {X 0,Y 383.244,Z 226.744,A -85,B 0,C 180,E1 -12156.317,E2 -12156.317} C_VEL
LIN {X 0,Y 383.136,Z 226.849,A -85,B 0,C 180,E1 -12159.569,E2 -12159.569} C_VEL
LIN {X 0,Y 385.192,Z 238.143,A -85,B 0,C 180,E1 -12162.479,E2 -12162.479} C_VEL
LIN {X 0,Y 388.984,Z 255.562,A -85,B 0,C 180,E1 -12163.026,E2 -12163.026} C_VEL
LIN {X 0,Y 390.083,Z 262.029,A -85,B 0,C 180,E1 -12163.21,E2 -12163.21} C_VEL
LIN {X 0,Y 388.59,Z 345.97,A -85,B 0,C 180,E1 -12164.834,E2 -12164.834} C_VEL
LIN {X 0,Y 388.108,Z 358.893,A -85,B 0,C 180,E1 -12165.289,E2 -12165.289} C_VEL
LIN {X 0,Y 387.958,Z 363.282,A -85,B 0,C 180,E1 -12165.495,E2 -12165.495} C_VEL
LIN {X 0,Y 386.952,Z 368.919,A -85,B 0,C 180,E1 -12165.763,E2 -12165.763} C_VEL
LIN {X 0,Y 383.684,Z 377.851,A -85,B 0,C 180,E1 -12166.218,E2 -12166.218} C_VEL
LIN {X 0,Y 380.422,Z 386.36,A -85,B 0,C 180,E1 -12166.775,E2 -12166.775} C_VEL
LIN {X 0,Y 379.444,Z 391.318,A -85,B 0,C 180,E1 -12167.203,E2 -12167.203} C_VEL
LIN {X 0,Y 378.506,Z 402.347,A -85,B 0,C 180,E1 -12168.4,E2 -12168.4} C_VEL
LIN {X 0,Y 377.447,Z 413.087,A -85,B 0,C 180,E1 -12169.865,E2 -12169.865} C_VEL
LIN {X 0,Y 376.764,Z 420.808,A -85,B 0,C 180,E1 -12171.169,E2 -12171.169} C_VEL
LIN {X 0,Y 376.02,Z 428.756,A -85,B 0,C 180,E1 -12172.819,E2 -12172.819} C_VEL
LIN {X 0,Y 375.454,Z 435.561,A -85,B 0,C 180,E1 -12174.612,E2 -12174.612} C_VEL
LIN {X 0,Y 375.038,Z 440.521,A -85,B 0,C 180,E1 -12176.29,E2 -12176.29} C_VEL
LIN {X 0,Y 374.783,Z 444.742,A -85,B 0,C 180,E1 -12178.213,E2 -12178.213} C_VEL
LIN {X 0,Y 374.431,Z 447.71,A -85,B 0,C 180,E1 -12180.316,E2 -12180.316} C_VEL
LIN {X 0,Y 374.316,Z 449.125,A -85,B 0,C 180,E1 -12182.356,E2 -12182.356} C_VEL
LIN {X 0,Y 374.318,Z 449.095,A -85,B 0,C 180,E1 -12184.314,E2 -12184.314} C_VEL
LIN {X 0,Y 374.477,Z 447.805,A -85,B 0,C 180,E1 -12186.211,E2 -12186.211} C_VEL
LIN {X 0,Y 374.792,Z 445.061,A -85,B 0,C 180,E1 -12188.228,E2 -12188.228} C_VEL
LIN {X 0,Y 375.247,Z 440.515,A -85,B 0,C 180,E1 -12190.339,E2 -12190.339} C_VEL
LIN {X 0,Y 375.678,Z 436.004,A -85,B 0,C 180,E1 -12191.886,E2 -12191.886} C_VEL
LIN {X 0,Y 376.396,Z 429.252,A -85,B 0,C 180,E1 -12193.697,E2 -12193.697} C_VEL
LIN {X 0,Y 377.112,Z 422.782,A -85,B 0,C 180,E1 -12195.085,E2 -12195.085} C_VEL
LIN {X 0,Y 378.058,Z 414.447,A -85,B 0,C 180,E1 -12196.554,E2 -12196.554} C_VEL
LIN {X 0,Y 379.029,Z 405.189,A -85,B 0,C 180,E1 -12197.873,E2 -12197.873} C_VEL
LIN {X 0,Y 380.057,Z 394.286,A -85,B 0,C 180,E1 -12199.126,E2 -12199.126} C_VEL
LIN {X 0,Y 381.058,Z 382.917,A -85,B 0,C 180,E1 -12200.159,E2 -12200.159} C_VEL
LIN {X 0,Y 381.853,Z 370.716,A -85,B 0,C 180,E1 -12201.011,E2 -12201.011} C_VEL
LIN {X 0,Y 382.567,Z 357.697,A -85,B 0,C 180,E1 -12201.673,E2 -12201.673} C_VEL
LIN {X 0,Y 383.015,Z 345.361,A -85,B 0,C 180,E1 -12202.091,E2 -12202.091} C_VEL
LIN {X 0,Y 384.605,Z 262.576,A -85,B 0,C 180,E1 -12203.739,E2 -12203.739} C_VEL
LIN {X 0,Y 381.004,Z 245.873,A -85,B 0,C 180,E1 -12204.327,E2 -12204.327} C_VEL
LIN {X 0,Y 378.346,Z 238.518,A -85,B 0,C 180,E1 -12204.685,E2 -12204.685} C_VEL
LIN {X 0,Y 375.954,Z 227.659,A -85,B 0,C 180,E1 -12207.482,E2 -12207.482} C_VEL
LIN {X 0,Y 375.978,Z 227.654,A -85,B 0,C 180,E1 -12211.465,E2 -12211.465} C_VEL
LIN {X 0,Y 375.976,Z 227.651,A -85,B 0,C 180,E1 -12214.545,E2 -12214.545} C_VEL
LIN {X 0,Y 375.936,Z 227.654,A -85,B 0,C 180,E1 -12218.052,E2 -12218.052} C_VEL
LIN {X 0,Y 375.984,Z 227.653,A -85,B 0,C 180,E1 -12221.48,E2 -12221.48} C_VEL
LIN {X 0,Y 376.038,Z 227.645,A -85,B 0,C 180,E1 -12224.839,E2 -12224.839} C_VEL
LIN {X 0,Y 376.04,Z 227.641,A -85,B 0,C 180,E1 -12228.143,E2 -12228.143} C_VEL
LIN {X 0,Y 376.183,Z 227.621,A -85,B 0,C 180,E1 -12231.947,E2 -12231.947} C_VEL
LIN {X 0,Y 376.146,Z 227.628,A -85,B 0,C 180,E1 -12234.646,E2 -12234.646} C_VEL
LIN {X 0,Y 376.338,Z 227.602,A -85,B 0,C 180,E1 -12237.866,E2 -12237.866} C_VEL
LIN {X 0,Y 376.473,Z 227.587,A -85,B 0,C 180,E1 -12240.006,E2 -12240.006} C_VEL
LIN {X 0,Y 376.33,Z 227.601,A -85,B 0,C 180,E1 -12242.146,E2 -12242.146} C_VEL
LIN {X 0,Y 376.211,Z 227.616,A -85,B 0,C 180,E1 -12246.441,E2 -12246.441} C_VEL
LIN {X 0,Y 376.106,Z 227.628,A -85,B 0,C 180,E1 -12249.687,E2 -12249.687} C_VEL
LIN {X 0,Y 376.088,Z 227.632,A -85,B 0,C 180,E1 -12253.663,E2 -12253.663} C_VEL
LIN {X 0,Y 376.032,Z 227.64,A -85,B 0,C 180,E1 -12257.405,E2 -12257.405} C_VEL
LIN {X 0,Y 375.981,Z 227.65,A -85,B 0,C 180,E1 -12260.837,E2 -12260.837} C_VEL
LIN {X 0,Y 375.937,Z 227.656,A -85,B 0,C 180,E1 -12264.29,E2 -12264.29} C_VEL
LIN {X 0,Y 375.914,Z 227.655,A -85,B 0,C 180,E1 -12266.665,E2 -12266.665} C_VEL
LIN {X 0,Y 375.918,Z 227.655,A -85,B 0,C 180,E1 -12269.089,E2 -12269.089} C_VEL
LIN {X 0,Y 375.943,Z 227.653,A -85,B 0,C 180,E1 -12271.568,E2 -12271.568} C_VEL
LIN {X 0,Y 375.981,Z 227.653,A -85,B 0,C 180,E1 -12274.67,E2 -12274.67} C_VEL
LIN {X 0,Y 375.938,Z 227.658,A -85,B 0,C 180,E1 -12278.266,E2 -12278.266} C_VEL
LIN {X 0,Y 375.918,Z 227.66,A -85,B 0,C 180,E1 -12281.6,E2 -12281.6} C_VEL
LIN {X 0,Y 375.905,Z 227.662,A -85,B 0,C 180,E1 -12285.277,E2 -12285.277} C_VEL
LIN {X 0,Y 375.922,Z 227.658,A -85,B 0,C 180,E1 -12289.132,E2 -12289.132} C_VEL
LIN {X 0,Y 375.959,Z 227.656,A -85,B 0,C 180,E1 -12291.912,E2 -12291.912} C_VEL
LIN {X 0,Y 375.986,Z 227.651,A -85,B 0,C 180,E1 -12295.337,E2 -12295.337} C_VEL
LIN {X 0,Y 375.947,Z 227.662,A -85,B 0,C 180,E1 -12298.438,E2 -12298.438} C_VEL
LIN {X 0,Y 375.997,Z 227.862,A -85,B 0,C 180,E1 -12300.31,E2 -12300.31} C_VEL
LIN {X 0,Y 378.635,Z 239.856,A -85,B 0,C 180,E1 -12303.259,E2 -12303.259} C_VEL
LIN {X 0,Y 379.847,Z 247.51,A -85,B 0,C 180,E1 -12305.047,E2 -12305.047} C_VEL
LIN {X 0,Y 378.776,Z 259.959,A -85,B 0,C 180,E1 -12307.702,E2 -12307.702} C_VEL
LIN {X 0,Y 378.535,Z 263.176,A -85,B 0,C 180,E1 -12308.384,E2 -12308.384} C_VEL
LIN {X 0,Y 382.62,Z 286.469,A -85,B 0,C 180,E1 -12309.151,E2 -12309.151} C_VEL
LIN {X 0,Y 384.085,Z 297.883,A -85,B 0,C 180,E1 -12309.481,E2 -12309.481} C_VEL
LIN {X 0,Y 382.722,Z 372.639,A -85,B 0,C 180,E1 -12310.978,E2 -12310.978} C_VEL
LIN {X 0,Y 382.038,Z 385.54,A -85,B 0,C 180,E1 -12311.429,E2 -12311.429} C_VEL
LIN {X 0,Y 381.185,Z 398.119,A -85,B 0,C 180,E1 -12312.082,E2 -12312.082} C_VEL
LIN {X 0,Y 380.155,Z 410.169,A -85,B 0,C 180,E1 -12312.934,E2 -12312.934} C_VEL
LIN {X 0,Y 379.077,Z 421.692,A -85,B 0,C 180,E1 -12313.992,E2 -12313.992} C_VEL
LIN {X 0,Y 378.094,Z 431.811,A -85,B 0,C 180,E1 -12315.155,E2 -12315.155} C_VEL
LIN {X 0,Y 377.157,Z 441.483,A -85,B 0,C 180,E1 -12316.531,E2 -12316.531} C_VEL
LIN {X 0,Y 376.152,Z 450.58,A -85,B 0,C 180,E1 -12318.14,E2 -12318.14} C_VEL
LIN {X 0,Y 375.457,Z 457.929,A -85,B 0,C 180,E1 -12319.757,E2 -12319.757} C_VEL
LIN {X 0,Y 375.008,Z 463.826,A -85,B 0,C 180,E1 -12321.378,E2 -12321.378} C_VEL
LIN {X 0,Y 374.696,Z 468.48,A -85,B 0,C 180,E1 -12322.997,E2 -12322.997} C_VEL
LIN {X 0,Y 374.53,Z 472.032,A -85,B 0,C 180,E1 -12324.617,E2 -12324.617} C_VEL
LIN {X 0,Y 374.529,Z 473.82,A -85,B 0,C 180,E1 -12325.696,E2 -12325.696} C_VEL
LIN {X 0,Y 374.504,Z 476.154,A -85,B 0,C 180,E1 -12327.849,E2 -12327.849} C_VEL
LIN {X 0,Y 374.549,Z 476.722,A -85,B 0,C 180,E1 -12328.925,E2 -12328.925} C_VEL
LIN {X 0,Y 374.583,Z 476.847,A -85,B 0,C 180,E1 -12330,E2 -12330} C_VEL
LIN {X 0,Y 374.564,Z 476.574,A -85,B 0,C 180,E1 -12331.075,E2 -12331.075} C_VEL
LIN {X 0,Y 374.508,Z 475.906,A -85,B 0,C 180,E1 -12332.151,E2 -12332.151} C_VEL
LIN {X 0,Y 374.473,Z 474.835,A -85,B 0,C 180,E1 -12333.228,E2 -12333.228} C_VEL
LIN {X 0,Y 374.555,Z 473.305,A -85,B 0,C 180,E1 -12334.304,E2 -12334.304} C_VEL
LIN {X 0,Y 374.586,Z 469.911,A -85,B 0,C 180,E1 -12336.048,E2 -12336.048} C_VEL
LIN {X 0,Y 374.779,Z 466.024,A -85,B 0,C 180,E1 -12337.543,E2 -12337.543} C_VEL
LIN {X 0,Y 375.166,Z 459.631,A -85,B 0,C 180,E1 -12339.434,E2 -12339.434} C_VEL
LIN {X 0,Y 375.688,Z 452.659,A -85,B 0,C 180,E1 -12341.055,E2 -12341.055} C_VEL
LIN {X 0,Y 376.54,Z 443.919,A -85,B 0,C 180,E1 -12342.668,E2 -12342.668} C_VEL
LIN {X 0,Y 377.33,Z 434.951,A -85,B 0,C 180,E1 -12344.012,E2 -12344.012} C_VEL
LIN {X 0,Y 378.133,Z 425.094,A -85,B 0,C 180,E1 -12345.22,E2 -12345.22} C_VEL
LIN {X 0,Y 379.041,Z 414.265,A -85,B 0,C 180,E1 -12346.286,E2 -12346.286} C_VEL
LIN {X 0,Y 379.981,Z 402.12,A -85,B 0,C 180,E1 -12347.213,E2 -12347.213} C_VEL
LIN {X 0,Y 380.812,Z 389.468,A -85,B 0,C 180,E1 -12347.937,E2 -12347.937} C_VEL
LIN {X 0,Y 381.454,Z 377.121,A -85,B 0,C 180,E1 -12348.426,E2 -12348.426} C_VEL
LIN {X 0,Y 381.817,Z 361.702,A -85,B 0,C 180,E1 -12348.791,E2 -12348.791} C_VEL
LIN {X 0,Y 382.805,Z 295.549,A -85,B 0,C 180,E1 -12350.081,E2 -12350.081} C_VEL
LIN {X 0,Y 378.082,Z 264.292,A -85,B 0,C 180,E1 -12350.989,E2 -12350.989} C_VEL
LIN {X 0,Y 379.435,Z 248.236,A -85,B 0,C 180,E1 -12354.458,E2 -12354.458} C_VEL
LIN {X 0,Y 379.436,Z 244.845,A -85,B 0,C 180,E1 -12355.214,E2 -12355.214} C_VEL
LIN {X 0,Y 376.946,Z 232.3,A -85,B 0,C 180,E1 -12358.215,E2 -12358.215} C_VEL
LIN {X 0,Y 375.969,Z 227.654,A -85,B 0,C 180,E1 -12359.385,E2 -12359.385} C_VEL
LIN {X 0,Y 375.927,Z 227.654,A -85,B 0,C 180,E1 -12362.83,E2 -12362.83} C_VEL
LIN {X 0,Y 375.94,Z 227.655,A -85,B 0,C 180,E1 -12365.416,E2 -12365.416} C_VEL
LIN {X 0,Y 375.938,Z 227.655,A -85,B 0,C 180,E1 -12368.258,E2 -12368.258} C_VEL
LIN {X 0,Y 375.903,Z 227.662,A -85,B 0,C 180,E1 -12371.59,E2 -12371.59} C_VEL
LIN {X 0,Y 375.895,Z 227.66,A -85,B 0,C 180,E1 -12375.272,E2 -12375.272} C_VEL
LIN {X 0,Y 375.916,Z 227.656,A -85,B 0,C 180,E1 -12378.401,E2 -12378.401} C_VEL
LIN {X 0,Y 375.955,Z 227.655,A -85,B 0,C 180,E1 -12381.905,E2 -12381.905} C_VEL
LIN {X 0,Y 375.979,Z 227.65,A -85,B 0,C 180,E1 -12385.331,E2 -12385.331} C_VEL
LIN {X 0,Y 375.94,Z 227.653,A -85,B 0,C 180,E1 -12388.431,E2 -12388.431} C_VEL
LIN {X 0,Y 375.952,Z 227.656,A -85,B 0,C 180,E1 -12391.473,E2 -12391.473} C_VEL
LIN {X 0,Y 375.939,Z 227.653,A -85,B 0,C 180,E1 -12394.529,E2 -12394.529} C_VEL
LIN {X 0,Y 375.973,Z 227.649,A -85,B 0,C 180,E1 -12396.882,E2 -12396.882} C_VEL
LIN {X 0,Y 375.964,Z 227.65,A -85,B 0,C 180,E1 -12400.332,E2 -12400.332} C_VEL
LIN {X 0,Y 376.012,Z 227.649,A -85,B 0,C 180,E1 -12403.713,E2 -12403.713} C_VEL
LIN {X 0,Y 376.099,Z 227.634,A -85,B 0,C 180,E1 -12407.036,E2 -12407.036} C_VEL
LIN {X 0,Y 376.072,Z 227.636,A -85,B 0,C 180,E1 -12410.312,E2 -12410.312} C_VEL
LIN {X 0,Y 376.148,Z 227.626,A -85,B 0,C 180,E1 -12412.479,E2 -12412.479} C_VEL
LIN {X 0,Y 376.132,Z 227.629,A -85,B 0,C 180,E1 -12414.634,E2 -12414.634} C_VEL
LIN {X 0,Y 376.319,Z 227.608,A -85,B 0,C 180,E1 -12417.853,E2 -12417.853} C_VEL
LIN {X 0,Y 376.328,Z 227.605,A -85,B 0,C 180,E1 -12422.134,E2 -12422.134} C_VEL
LIN {X 0,Y 376.171,Z 227.624,A -85,B 0,C 180,E1 -12426.457,E2 -12426.457} C_VEL
LIN {X 0,Y 376.092,Z 227.638,A -85,B 0,C 180,E1 -12429.675,E2 -12429.675} C_VEL
LIN {X 0,Y 376.07,Z 227.641,A -85,B 0,C 180,E1 -12433.651,E2 -12433.651} C_VEL
LIN {X 0,Y 376.01,Z 227.65,A -85,B 0,C 180,E1 -12437.393,E2 -12437.393} C_VEL
LIN {X 0,Y 375.953,Z 227.652,A -85,B 0,C 180,E1 -12440.826,E2 -12440.826} C_VEL
LIN {X 0,Y 375.949,Z 227.651,A -85,B 0,C 180,E1 -12444.276,E2 -12444.276} C_VEL
LIN {X 0,Y 375.945,Z 227.654,A -85,B 0,C 180,E1 -12447.854,E2 -12447.854} C_VEL
LIN {X 0,Y 375.922,Z 227.659,A -85,B 0,C 180,E1 -12451.556,E2 -12451.556} C_VEL
LIN {X 0,Y 375.919,Z 227.661,A -85,B 0,C 180,E1 -12455.41,E2 -12455.41} C_VEL
LIN {X 0,Y 375.934,Z 227.653,A -85,B 0,C 180,E1 -12458.264,E2 -12458.264} C_VEL
LIN {X 0,Y 375.892,Z 227.662,A -85,B 0,C 180,E1 -12461.595,E2 -12461.595} C_VEL
LIN {X 0,Y 375.908,Z 227.663,A -85,B 0,C 180,E1 -12465.26,E2 -12465.26} C_VEL
LIN {X 0,Y 375.891,Z 227.664,A -85,B 0,C 180,E1 -12469.128,E2 -12469.128} C_VEL
LIN {X 0,Y 375.915,Z 227.656,A -85,B 0,C 180,E1 -12471.907,E2 -12471.907} C_VEL
LIN {X 0,Y 375.928,Z 227.659,A -85,B 0,C 180,E1 -12475.328,E2 -12475.328} C_VEL
LIN {X 0,Y 375.906,Z 227.657,A -85,B 0,C 180,E1 -12478.434,E2 -12478.434} C_VEL
LIN {X 0,Y 375.947,Z 227.652,A -85,B 0,C 180,E1 -12482.138,E2 -12482.138} C_VEL
LIN {X 0,Y 375.951,Z 227.652,A -85,B 0,C 180,E1 -12484.536,E2 -12484.536} C_VEL
LIN {X 0,Y 375.962,Z 227.65,A -85,B 0,C 180,E1 -12488.046,E2 -12488.046} C_VEL
LIN {X 0,Y 375.973,Z 227.651,A -85,B 0,C 180,E1 -12491.472,E2 -12491.472} C_VEL
LIN {X 0,Y 376.002,Z 227.648,A -85,B 0,C 180,E1 -12494.831,E2 -12494.831} C_VEL
LIN {X 0,Y 375.999,Z 227.645,A -85,B 0,C 180,E1 -12498.135,E2 -12498.135} C_VEL
LIN {X 0,Y 376.204,Z 227.62,A -85,B 0,C 180,E1 -12501.869,E2 -12501.869} C_VEL
LIN {X 0,Y 376.121,Z 227.632,A -85,B 0,C 180,E1 -12504.639,E2 -12504.639} C_VEL
LIN {X 0,Y 376.296,Z 227.608,A -85,B 0,C 180,E1 -12507.859,E2 -12507.859} C_VEL
LIN {X 0,Y 376.429,Z 227.592,A -85,B 0,C 180,E1 -12510,E2 -12510} C_VEL
LIN {X 0,Y 376.157,Z 227.63,A -85,B 0,C 180,E1 -12513.213,E2 -12513.213} C_VEL
LIN {X 0,Y 376.201,Z 227.622,A -85,B 0,C 180,E1 -12516.436,E2 -12516.436} C_VEL
LIN {X 0,Y 376.08,Z 227.733,A -85,B 0,C 180,E1 -12519.309,E2 -12519.309} C_VEL
LIN {X 0,Y 378.154,Z 238.517,A -85,B 0,C 180,E1 -12522.116,E2 -12522.116} C_VEL
LIN {X 0,Y 380.392,Z 247.172,A -85,B 0,C 180,E1 -12522.414,E2 -12522.414} C_VEL
LIN {X 0,Y 383.329,Z 262.371,A -85,B 0,C 180,E1 -12522.878,E2 -12522.878} C_VEL
LIN {X 0,Y 381.825,Z 345.939,A -85,B 0,C 180,E1 -12524.524,E2 -12524.524} C_VEL
LIN {X 0,Y 381.305,Z 358.99,A -85,B 0,C 180,E1 -12524.987,E2 -12524.987} C_VEL
LIN {X 0,Y 380.739,Z 371.718,A -85,B 0,C 180,E1 -12525.661,E2 -12525.661} C_VEL
LIN {X 0,Y 379.993,Z 383.631,A -85,B 0,C 180,E1 -12526.52,E2 -12526.52} C_VEL
LIN {X 0,Y 379.444,Z 391.318,A -85,B 0,C 180,E1 -12527.203,E2 -12527.203} C_VEL
LIN {X 0,Y 378.41,Z 396.271,A -85,B 0,C 180,E1 -12527.668,E2 -12527.668} C_VEL
LIN {X 0,Y 374.872,Z 404.013,A -85,B 0,C 180,E1 -12528.449,E2 -12528.449} C_VEL
LIN {X 0,Y 371.328,Z 411.231,A -85,B 0,C 180,E1 -12529.343,E2 -12529.343} C_VEL
LIN {X 0,Y 370.297,Z 415.36,A -85,B 0,C 180,E1 -12529.976,E2 -12529.976} C_VEL
LIN {X 0,Y 369.545,Z 423.738,A -85,B 0,C 180,E1 -12531.507,E2 -12531.507} C_VEL
LIN {X 0,Y 368.888,Z 430.366,A -85,B 0,C 180,E1 -12532.989,E2 -12532.989} C_VEL
LIN {X 0,Y 368.286,Z 436.929,A -85,B 0,C 180,E1 -12534.823,E2 -12534.823} C_VEL
LIN {X 0,Y 367.899,Z 441.967,A -85,B 0,C 180,E1 -12536.683,E2 -12536.683} C_VEL
LIN {X 0,Y 367.633,Z 445.656,A -85,B 0,C 180,E1 -12538.549,E2 -12538.549} C_VEL
LIN {X 0,Y 367.307,Z 448.276,A -85,B 0,C 180,E1 -12540.586,E2 -12540.586} C_VEL
LIN {X 0,Y 367.224,Z 449.447,A -85,B 0,C 180,E1 -12542.656,E2 -12542.656} C_VEL
LIN {X 0,Y 367.229,Z 449.248,A -85,B 0,C 180,E1 -12544.637,E2 -12544.637} C_VEL
LIN {X 0,Y 367.437,Z 447.81,A -85,B 0,C 180,E1 -12546.565,E2 -12546.565} C_VEL
LIN {X 0,Y 367.754,Z 445.218,A -85,B 0,C 180,E1 -12548.429,E2 -12548.429} C_VEL
LIN {X 0,Y 368.211,Z 440.91,A -85,B 0,C 180,E1 -12550.461,E2 -12550.461} C_VEL
LIN {X 0,Y 368.631,Z 436.627,A -85,B 0,C 180,E1 -12551.979,E2 -12551.979} C_VEL
LIN {X 0,Y 369.328,Z 430.452,A -85,B 0,C 180,E1 -12553.701,E2 -12553.701} C_VEL
LIN {X 0,Y 370.227,Z 422.806,A -85,B 0,C 180,E1 -12555.395,E2 -12555.395} C_VEL
LIN {X 0,Y 371.177,Z 415.007,A -85,B 0,C 180,E1 -12556.79,E2 -12556.79} C_VEL
LIN {X 0,Y 372.098,Z 406.515,A -85,B 0,C 180,E1 -12558.045,E2 -12558.045} C_VEL
LIN {X 0,Y 373.139,Z 396.077,A -85,B 0,C 180,E1 -12559.295,E2 -12559.295} C_VEL
LIN {X 0,Y 374.18,Z 384.937,A -85,B 0,C 180,E1 -12560.359,E2 -12560.359} C_VEL
LIN {X 0,Y 375.052,Z 372.907,A -85,B 0,C 180,E1 -12561.258,E2 -12561.258} C_VEL
LIN {X 0,Y 375.823,Z 360.139,A -85,B 0,C 180,E1 -12561.951,E2 -12561.951} C_VEL
LIN {X 0,Y 376.345,Z 346.929,A -85,B 0,C 180,E1 -12562.439,E2 -12562.439} C_VEL
LIN {X 0,Y 378.102,Z 263.731,A -85,B 0,C 180,E1 -12564.135,E2 -12564.135} C_VEL
LIN {X 0,Y 374.564,Z 247.355,A -85,B 0,C 180,E1 -12564.728,E2 -12564.728} C_VEL
LIN {X 0,Y 371.179,Z 238.787,A -85,B 0,C 180,E1 -12565.181,E2 -12565.181} C_VEL
LIN {X 0,Y 368.892,Z 228.538,A -85,B 0,C 180,E1 -12567.904,E2 -12567.904} C_VEL
LIN {X 0,Y 368.955,Z 228.528,A -85,B 0,C 180,E1 -12571.571,E2 -12571.571} C_VEL
LIN {X 0,Y 368.928,Z 228.531,A -85,B 0,C 180,E1 -12575.231,E2 -12575.231} C_VEL
LIN {X 0,Y 368.912,Z 228.537,A -85,B 0,C 180,E1 -12578.98,E2 -12578.98} C_VEL
LIN {X 0,Y 368.968,Z 228.526,A -85,B 0,C 180,E1 -12582.264,E2 -12582.264} C_VEL
LIN {X 0,Y 369.018,Z 228.517,A -85,B 0,C 180,E1 -12586.234,E2 -12586.234} C_VEL
LIN {X 0,Y 369.049,Z 228.514,A -85,B 0,C 180,E1 -12590.138,E2 -12590.138} C_VEL
LIN {X 0,Y 369.165,Z 228.499,A -85,B 0,C 180,E1 -12593.448,E2 -12593.448} C_VEL
LIN {X 0,Y 369.303,Z 228.478,A -85,B 0,C 180,E1 -12597.825,E2 -12597.825} C_VEL
LIN {X 0,Y 369.443,Z 228.463,A -85,B 0,C 180,E1 -12600.006,E2 -12600.006} C_VEL
LIN {X 0,Y 369.294,Z 228.477,A -85,B 0,C 180,E1 -12602.187,E2 -12602.187} C_VEL
LIN {X 0,Y 369.172,Z 228.493,A -85,B 0,C 180,E1 -12606.565,E2 -12606.565} C_VEL
LIN {X 0,Y 369.056,Z 228.506,A -85,B 0,C 180,E1 -12609.874,E2 -12609.874} C_VEL
LIN {X 0,Y 369.036,Z 228.51,A -85,B 0,C 180,E1 -12613.777,E2 -12613.777} C_VEL
LIN {X 0,Y 368.992,Z 228.517,A -85,B 0,C 180,E1 -12617.748,E2 -12617.748} C_VEL
LIN {X 0,Y 368.911,Z 228.528,A -85,B 0,C 180,E1 -12621.226,E2 -12621.226} C_VEL
LIN {X 0,Y 368.91,Z 228.528,A -85,B 0,C 180,E1 -12623.878,E2 -12623.878} C_VEL
LIN {X 0,Y 368.861,Z 228.534,A -85,B 0,C 180,E1 -12627.217,E2 -12627.217} C_VEL
LIN {X 0,Y 368.898,Z 228.528,A -85,B 0,C 180,E1 -12629.697,E2 -12629.697} C_VEL
LIN {X 0,Y 368.901,Z 228.526,A -85,B 0,C 180,E1 -12633.543,E2 -12633.543} C_VEL
LIN {X 0,Y 368.901,Z 228.53,A -85,B 0,C 180,E1 -12636.858,E2 -12636.858} C_VEL
LIN {X 0,Y 368.892,Z 228.534,A -85,B 0,C 180,E1 -12640.378,E2 -12640.378} C_VEL
LIN {X 0,Y 368.863,Z 228.54,A -85,B 0,C 180,E1 -12643.614,E2 -12643.614} C_VEL
LIN {X 0,Y 368.855,Z 228.541,A -85,B 0,C 180,E1 -12646.693,E2 -12646.693} C_VEL
LIN {X 0,Y 368.895,Z 228.534,A -85,B 0,C 180,E1 -12649.652,E2 -12649.652} C_VEL
LIN {X 0,Y 368.905,Z 228.533,A -85,B 0,C 180,E1 -12653.149,E2 -12653.149} C_VEL
LIN {X 0,Y 368.907,Z 228.535,A -85,B 0,C 180,E1 -12656.464,E2 -12656.464} C_VEL
LIN {X 0,Y 368.947,Z 228.677,A -85,B 0,C 180,E1 -12659.881,E2 -12659.881} C_VEL
LIN {X 0,Y 371.481,Z 240.135,A -85,B 0,C 180,E1 -12662.778,E2 -12662.778} C_VEL
LIN {X 0,Y 372.972,Z 248.35,A -85,B 0,C 180,E1 -12664.76,E2 -12664.76} C_VEL
LIN {X 0,Y 372.009,Z 259.615,A -85,B 0,C 180,E1 -12667.215,E2 -12667.215} C_VEL
LIN {X 0,Y 371.699,Z 262.865,A -85,B 0,C 180,E1 -12667.915,E2 -12667.915} C_VEL
LIN {X 0,Y 375.788,Z 285.343,A -85,B 0,C 180,E1 -12668.689,E2 -12668.689} C_VEL
LIN {X 0,Y 377.525,Z 298.21,A -85,B 0,C 180,E1 -12669.079,E2 -12669.079} C_VEL
LIN {X 0,Y 376.076,Z 372.291,A -85,B 0,C 180,E1 -12670.593,E2 -12670.593} C_VEL
LIN {X 0,Y 375.369,Z 385.187,A -85,B 0,C 180,E1 -12671.052,E2 -12671.052} C_VEL
LIN {X 0,Y 374.438,Z 398.323,A -85,B 0,C 180,E1 -12671.747,E2 -12671.747} C_VEL
LIN {X 0,Y 373.376,Z 410.237,A -85,B 0,C 180,E1 -12672.614,E2 -12672.614} C_VEL
LIN {X 0,Y 372.237,Z 421.7,A -85,B 0,C 180,E1 -12673.69,E2 -12673.69} C_VEL
LIN {X 0,Y 371.125,Z 432.598,A -85,B 0,C 180,E1 -12674.981,E2 -12674.981} C_VEL
LIN {X 0,Y 370.233,Z 441.391,A -85,B 0,C 180,E1 -12676.274,E2 -12676.274} C_VEL
LIN {X 0,Y 369.206,Z 450.462,A -85,B 0,C 180,E1 -12677.914,E2 -12677.914} C_VEL
LIN {X 0,Y 368.454,Z 457.786,A -85,B 0,C 180,E1 -12679.56,E2 -12679.56} C_VEL
LIN {X 0,Y 367.974,Z 463.657,A -85,B 0,C 180,E1 -12681.211,E2 -12681.211} C_VEL
LIN {X 0,Y 367.62,Z 468.288,A -85,B 0,C 180,E1 -12682.862,E2 -12682.862} C_VEL
LIN {X 0,Y 367.444,Z 471.82,A -85,B 0,C 180,E1 -12684.512,E2 -12684.512} C_VEL
LIN {X 0,Y 367.436,Z 473.593,A -85,B 0,C 180,E1 -12685.612,E2 -12685.612} C_VEL
LIN {X 0,Y 367.403,Z 475.91,A -85,B 0,C 180,E1 -12687.808,E2 -12687.808} C_VEL
LIN {X 0,Y 367.451,Z 476.465,A -85,B 0,C 180,E1 -12688.904,E2 -12688.904} C_VEL
LIN {X 0,Y 367.5,Z 476.581,A -85,B 0,C 180,E1 -12690,E2 -12690} C_VEL
LIN {X 0,Y 367.466,Z 476.299,A -85,B 0,C 180,E1 -12691.096,E2 -12691.096} C_VEL
LIN {X 0,Y 367.408,Z 475.624,A -85,B 0,C 180,E1 -12692.193,E2 -12692.193} C_VEL
LIN {X 0,Y 367.391,Z 474.539,A -85,B 0,C 180,E1 -12693.29,E2 -12693.29} C_VEL
LIN {X 0,Y 367.459,Z 472.996,A -85,B 0,C 180,E1 -12694.388,E2 -12694.388} C_VEL
LIN {X 0,Y 367.483,Z 469.973,A -85,B 0,C 180,E1 -12695.994,E2 -12695.994} C_VEL
LIN {X 0,Y 367.707,Z 465.674,A -85,B 0,C 180,E1 -12697.689,E2 -12697.689} C_VEL
LIN {X 0,Y 368.132,Z 459.255,A -85,B 0,C 180,E1 -12699.616,E2 -12699.616} C_VEL
LIN {X 0,Y 368.682,Z 452.247,A -85,B 0,C 180,E1 -12701.267,E2 -12701.267} C_VEL
LIN {X 0,Y 369.571,Z 443.457,A -85,B 0,C 180,E1 -12702.911,E2 -12702.911} C_VEL
LIN {X 0,Y 370.41,Z 434.442,A -85,B 0,C 180,E1 -12704.279,E2 -12704.279} C_VEL
LIN {X 0,Y 371.238,Z 424.525,A -85,B 0,C 180,E1 -12705.509,E2 -12705.509} C_VEL
LIN {X 0,Y 372.178,Z 413.579,A -85,B 0,C 180,E1 -12706.595,E2 -12706.595} C_VEL
LIN {X 0,Y 373.181,Z 401.322,A -85,B 0,C 180,E1 -12707.537,E2 -12707.537} C_VEL
LIN {X 0,Y 374.061,Z 388.485,A -85,B 0,C 180,E1 -12708.272,E2 -12708.272} C_VEL
LIN {X 0,Y 374.694,Z 375.634,A -85,B 0,C 180,E1 -12708.771,E2 -12708.771} C_VEL
LIN {X 0,Y 375.152,Z 356.137,A -85,B 0,C 180,E1 -12709.208,E2 -12709.208} C_VEL
LIN {X 0,Y 376.02,Z 296.14,A -85,B 0,C 180,E1 -12710.404,E2 -12710.404} C_VEL
LIN {X 0,Y 371.163,Z 264.129,A -85,B 0,C 180,E1 -12711.342,E2 -12711.342} C_VEL
LIN {X 0,Y 372.446,Z 249.66,A -85,B 0,C 180,E1 -12714.527,E2 -12714.527} C_VEL
LIN {X 0,Y 372.483,Z 246.086,A -85,B 0,C 180,E1 -12715.338,E2 -12715.338} C_VEL
LIN {X 0,Y 369.679,Z 232.025,A -85,B 0,C 180,E1 -12718.774,E2 -12718.774} C_VEL
LIN {X 0,Y 368.93,Z 228.532,A -85,B 0,C 180,E1 -12719.688,E2 -12719.688} C_VEL
LIN {X 0,Y 368.878,Z 228.536,A -85,B 0,C 180,E1 -12723.539,E2 -12723.539} C_VEL
LIN {X 0,Y 368.901,Z 228.529,A -85,B 0,C 180,E1 -12726.85,E2 -12726.85} C_VEL
LIN {X 0,Y 368.895,Z 228.531,A -85,B 0,C 180,E1 -12730.371,E2 -12730.371} C_VEL
LIN {X 0,Y 368.845,Z 228.541,A -85,B 0,C 180,E1 -12733.604,E2 -12733.604} C_VEL
LIN {X 0,Y 368.852,Z 228.535,A -85,B 0,C 180,E1 -12736.686,E2 -12736.686} C_VEL
LIN {X 0,Y 368.894,Z 228.536,A -85,B 0,C 180,E1 -12739.645,E2 -12739.645} C_VEL
LIN {X 0,Y 368.898,Z 228.531,A -85,B 0,C 180,E1 -12743.143,E2 -12743.143} C_VEL
LIN {X 0,Y 368.901,Z 228.53,A -85,B 0,C 180,E1 -12746.457,E2 -12746.457} C_VEL
LIN {X 0,Y 368.896,Z 228.531,A -85,B 0,C 180,E1 -12750.303,E2 -12750.303} C_VEL
LIN {X 0,Y 368.922,Z 228.529,A -85,B 0,C 180,E1 -12754.009,E2 -12754.009} C_VEL
LIN {X 0,Y 368.919,Z 228.534,A -85,B 0,C 180,E1 -12757.599,E2 -12757.599} C_VEL
LIN {X 0,Y 368.912,Z 228.53,A -85,B 0,C 180,E1 -12761.098,E2 -12761.098} C_VEL
LIN {X 0,Y 368.987,Z 228.519,A -85,B 0,C 180,E1 -12764.529,E2 -12764.529} C_VEL
LIN {X 0,Y 369.055,Z 228.51,A -85,B 0,C 180,E1 -12766.785,E2 -12766.785} C_VEL
LIN {X 0,Y 369.032,Z 228.514,A -85,B 0,C 180,E1 -12770.125,E2 -12770.125} C_VEL
LIN {X 0,Y 369.148,Z 228.504,A -85,B 0,C 180,E1 -12773.435,E2 -12773.435} C_VEL
LIN {X 0,Y 369.282,Z 228.485,A -85,B 0,C 180,E1 -12777.813,E2 -12777.813} C_VEL
LIN {X 0,Y 369.292,Z 228.481,A -85,B 0,C 180,E1 -12782.175,E2 -12782.175} C_VEL
LIN {X 0,Y 369.136,Z 228.5,A -85,B 0,C 180,E1 -12786.553,E2 -12786.553} C_VEL
LIN {X 0,Y 369.042,Z 228.514,A -85,B 0,C 180,E1 -12789.862,E2 -12789.862} C_VEL
LIN {X 0,Y 369.018,Z 228.518,A -85,B 0,C 180,E1 -12793.765,E2 -12793.765} C_VEL
LIN {X 0,Y 368.968,Z 228.524,A -85,B 0,C 180,E1 -12797.736,E2 -12797.736} C_VEL
LIN {X 0,Y 368.904,Z 228.534,A -85,B 0,C 180,E1 -12801.213,E2 -12801.213} C_VEL
LIN {X 0,Y 368.91,Z 228.529,A -85,B 0,C 180,E1 -12804.77,E2 -12804.77} C_VEL
LIN {X 0,Y 368.928,Z 228.526,A -85,B 0,C 180,E1 -12808.432,E2 -12808.432} C_VEL
LIN {X 0,Y 368.863,Z 228.534,A -85,B 0,C 180,E1 -12812.232,E2 -12812.232} C_VEL
LIN {X 0,Y 368.892,Z 228.534,A -85,B 0,C 180,E1 -12814.995,E2 -12814.995} C_VEL
LIN {X 0,Y 368.868,Z 228.534,A -85,B 0,C 180,E1 -12818.634,E2 -12818.634} C_VEL
LIN {X 0,Y 368.839,Z 228.538,A -85,B 0,C 180,E1 -12822.004,E2 -12822.004} C_VEL
LIN {X 0,Y 368.881,Z 228.537,A -85,B 0,C 180,E1 -12825.177,E2 -12825.177} C_VEL
LIN {X 0,Y 368.835,Z 228.538,A -85,B 0,C 180,E1 -12828.172,E2 -12828.172} C_VEL
LIN {X 0,Y 368.86,Z 228.54,A -85,B 0,C 180,E1 -12831.355,E2 -12831.355} C_VEL
LIN {X 0,Y 368.885,Z 228.537,A -85,B 0,C 180,E1 -12835.142,E2 -12835.142} C_VEL
LIN {X 0,Y 368.877,Z 228.537,A -85,B 0,C 180,E1 -12839.042,E2 -12839.042} C_VEL
LIN {X 0,Y 368.932,Z 228.528,A -85,B 0,C 180,E1 -12841.561,E2 -12841.561} C_VEL
LIN {X 0,Y 368.905,Z 228.535,A -85,B 0,C 180,E1 -12845.222,E2 -12845.222} C_VEL
LIN {X 0,Y 368.918,Z 228.532,A -85,B 0,C 180,E1 -12848.955,E2 -12848.955} C_VEL
LIN {X 0,Y 368.934,Z 228.525,A -85,B 0,C 180,E1 -12852.255,E2 -12852.255} C_VEL
LIN {X 0,Y 368.978,Z 228.52,A -85,B 0,C 180,E1 -12856.226,E2 -12856.226} C_VEL
LIN {X 0,Y 369.014,Z 228.515,A -85,B 0,C 180,E1 -12860.13,E2 -12860.13} C_VEL
LIN {X 0,Y 369.141,Z 228.5,A -85,B 0,C 180,E1 -12862.341,E2 -12862.341} C_VEL
LIN {X 0,Y 369.094,Z 228.507,A -85,B 0,C 180,E1 -12864.537,E2 -12864.537} C_VEL
LIN {X 0,Y 369.262,Z 228.485,A -85,B 0,C 180,E1 -12867.818,E2 -12867.818} C_VEL
LIN {X 0,Y 369.399,Z 228.467,A -85,B 0,C 180,E1 -12870,E2 -12870} C_VEL
LIN {X 0,Y 369.262,Z 228.484,A -85,B 0,C 180,E1 -12872.181,E2 -12872.181} C_VEL
LIN {X 0,Y 369.16,Z 228.499,A -85,B 0,C 180,E1 -12876.559,E2 -12876.559} C_VEL
LIN {X 0,Y 369.07,Z 228.591,A -85,B 0,C 180,E1 -12879.038,E2 -12879.038} C_VEL
LIN {X 0,Y 370.937,Z 238.494,A -85,B 0,C 180,E1 -12881.717,E2 -12881.717} C_VEL
LIN {X 0,Y 373.405,Z 247.04,A -85,B 0,C 180,E1 -12882.04,E2 -12882.04} C_VEL
LIN {X 0,Y 376.467,Z 262.562,A -85,B 0,C 180,E1 -12882.53,E2 -12882.53} C_VEL
LIN {X 0,Y 375.04,Z 345.781,A -85,B 0,C 180,E1 -12884.203,E2 -12884.203} C_VEL
LIN {X 0,Y 374.504,Z 359.704,A -85,B 0,C 180,E1 -12884.71,E2 -12884.71} C_VEL
LIN {X 0,Y 373.916,Z 372.133,A -85,B 0,C 180,E1 -12885.385,E2 -12885.385} C_VEL
LIN {X 0,Y 373.105,Z 384.538,A -85,B 0,C 180,E1 -12886.304,E2 -12886.304} C_VEL
LIN {X 0,Y 372.124,Z 396.465,A -85,B 0,C 180,E1 -12887.446,E2 -12887.446} C_VEL
LIN {X 0,Y 371.185,Z 406.649,A -85,B 0,C 180,E1 -12888.68,E2 -12888.68} C_VEL
LIN {X 0,Y 370.297,Z 415.36,A -85,B 0,C 180,E1 -12889.976,E2 -12889.976} C_VEL
LIN {X 0,Y 369.286,Z 419.357,A -85,B 0,C 180,E1 -12890.64,E2 -12890.64} C_VEL
LIN {X 0,Y 365.822,Z 425.446,A -85,B 0,C 180,E1 -12891.736,E2 -12891.736} C_VEL
LIN {X 0,Y 362.429,Z 430.942,A -85,B 0,C 180,E1 -12892.922,E2 -12892.922} C_VEL
LIN {X 0,Y 361.542,Z 433.936,A -85,B 0,C 180,E1 -12893.715,E2 -12893.715} C_VEL
LIN {X 0,Y 361.058,Z 439.094,A -85,B 0,C 180,E1 -12895.354,E2 -12895.354} C_VEL
LIN {X 0,Y 360.753,Z 443.653,A -85,B 0,C 180,E1 -12897.245,E2 -12897.245} C_VEL
LIN {X 0,Y 360.4,Z 446.931,A -85,B 0,C 180,E1 -12899.176,E2 -12899.176} C_VEL
LIN {X 0,Y 360.186,Z 448.773,A -85,B 0,C 180,E1 -12900.866,E2 -12900.866} C_VEL
LIN {X 0,Y 360.131,Z 449.783,A -85,B 0,C 180,E1 -12903.121,E2 -12903.121} C_VEL
LIN {X 0,Y 360.153,Z 449.403,A -85,B 0,C 180,E1 -12904.973,E2 -12904.973} C_VEL
LIN {X 0,Y 360.441,Z 447.481,A -85,B 0,C 180,E1 -12907.188,E2 -12907.188} C_VEL
LIN {X 0,Y 360.864,Z 444.037,A -85,B 0,C 180,E1 -12909.353,E2 -12909.353} C_VEL
LIN {X 0,Y 361.38,Z 439.222,A -85,B 0,C 180,E1 -12911.392,E2 -12911.392} C_VEL
LIN {X 0,Y 362.046,Z 433.662,A -85,B 0,C 180,E1 -12913.154,E2 -12913.154} C_VEL
LIN {X 0,Y 362.938,Z 426.363,A -85,B 0,C 180,E1 -12914.973,E2 -12914.973} C_VEL
LIN {X 0,Y 363.837,Z 418.855,A -85,B 0,C 180,E1 -12916.475,E2 -12916.475} C_VEL
LIN {X 0,Y 365.035,Z 409.132,A -85,B 0,C 180,E1 -12918.034,E2 -12918.034} C_VEL
LIN {X 0,Y 366.163,Z 398.92,A -85,B 0,C 180,E1 -12919.352,E2 -12919.352} C_VEL
LIN {X 0,Y 367.265,Z 387.531,A -85,B 0,C 180,E1 -12920.521,E2 -12920.521} C_VEL
LIN {X 0,Y 368.26,Z 375.395,A -85,B 0,C 180,E1 -12921.484,E2 -12921.484} C_VEL
LIN {X 0,Y 369.056,Z 363.268,A -85,B 0,C 180,E1 -12922.208,E2 -12922.208} C_VEL
LIN {X 0,Y 369.629,Z 350.64,A -85,B 0,C 180,E1 -12922.733,E2 -12922.733} C_VEL
LIN {X 0,Y 370.113,Z 333.352,A -85,B 0,C 180,E1 -12923.147,E2 -12923.147} C_VEL
LIN {X 0,Y 371.499,Z 264.283,A -85,B 0,C 180,E1 -12924.566,E2 -12924.566} C_VEL
LIN {X 0,Y 368.413,Z 250.05,A -85,B 0,C 180,E1 -12925.1,E2 -12925.1} C_VEL
LIN {X 0,Y 364.061,Z 239.184,A -85,B 0,C 180,E1 -12925.673,E2 -12925.673} C_VEL
LIN {X 0,Y 361.844,Z 229.415,A -85,B 0,C 180,E1 -12928.34,E2 -12928.34} C_VEL
LIN {X 0,Y 361.891,Z 229.406,A -85,B 0,C 180,E1 -12932.228,E2 -12932.228} C_VEL
LIN {X 0,Y 361.899,Z 229.407,A -85,B 0,C 180,E1 -12934.716,E2 -12934.716} C_VEL
LIN {X 0,Y 361.866,Z 229.409,A -85,B 0,C 180,E1 -12938.354,E2 -12938.354} C_VEL
LIN {X 0,Y 361.944,Z 229.401,A -85,B 0,C 180,E1 -12942.068,E2 -12942.068} C_VEL
LIN {X 0,Y 361.978,Z 229.393,A -85,B 0,C 180,E1 -12946.108,E2 -12946.108} C_VEL
LIN {X 0,Y 362.014,Z 229.39,A -85,B 0,C 180,E1 -12949.944,E2 -12949.944} C_VEL
LIN {X 0,Y 362.127,Z 229.376,A -85,B 0,C 180,E1 -12953.32,E2 -12953.32} C_VEL
LIN {X 0,Y 362.267,Z 229.355,A -85,B 0,C 180,E1 -12957.783,E2 -12957.783} C_VEL
LIN {X 0,Y 362.392,Z 229.342,A -85,B 0,C 180,E1 -12960.006,E2 -12960.006} C_VEL
LIN {X 0,Y 362.257,Z 229.354,A -85,B 0,C 180,E1 -12962.23,E2 -12962.23} C_VEL
LIN {X 0,Y 362.134,Z 229.37,A -85,B 0,C 180,E1 -12966.693,E2 -12966.693} C_VEL
LIN {X 0,Y 361.993,Z 229.386,A -85,B 0,C 180,E1 -12970.069,E2 -12970.069} C_VEL
LIN {X 0,Y 361.997,Z 229.387,A -85,B 0,C 180,E1 -12973.904,E2 -12973.904} C_VEL
LIN {X 0,Y 361.928,Z 229.4,A -85,B 0,C 180,E1 -12976.94,E2 -12976.94} C_VEL
LIN {X 0,Y 361.885,Z 229.408,A -85,B 0,C 180,E1 -12980.466,E2 -12980.466} C_VEL
LIN {X 0,Y 361.865,Z 229.407,A -85,B 0,C 180,E1 -12984.106,E2 -12984.106} C_VEL
LIN {X 0,Y 361.839,Z 229.409,A -85,B 0,C 180,E1 -12987.79,E2 -12987.79} C_VEL
LIN {X 0,Y 361.832,Z 229.411,A -85,B 0,C 180,E1 -12991.284,E2 -12991.284} C_VEL
LIN {X 0,Y 361.857,Z 229.407,A -85,B 0,C 180,E1 -12994.285,E2 -12994.285} C_VEL
LIN {X 0,Y 361.863,Z 229.407,A -85,B 0,C 180,E1 -12997.225,E2 -12997.225} C_VEL
LIN {X 0,Y 361.818,Z 229.419,A -85,B 0,C 180,E1 -13000.754,E2 -13000.754} C_VEL
LIN {X 0,Y 361.801,Z 229.421,A -85,B 0,C 180,E1 -13004.376,E2 -13004.376} C_VEL
LIN {X 0,Y 361.821,Z 229.416,A -85,B 0,C 180,E1 -13007.576,E2 -13007.576} C_VEL
